KUKA KRL program: Milling_8_3.src

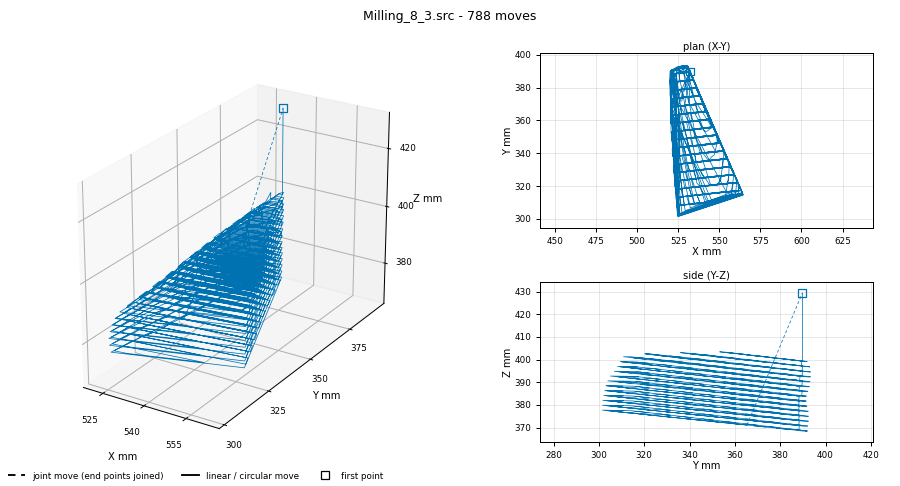
[picture p0: tool path of Milling_8_3.src, 788 of 790 moves have a stored position in this frame; points joined in program order, loops and branches not executed]
&ACCESS RVP
&REL 1
&PARAM TEMPLATE = C:\KRC\Roboter\Template\vorgabe
&PARAM EDITMASK = *
DEF Milling_8_3 ( )


;FOLD INI
;FOLD BASISTECH INI
GLOBAL INTERRUPT DECL 3 WHEN $STOPMESS==TRUE DO IR_STOPM ( )
INTERRUPT ON 3
BAS (#INITMOV,0 )
;ENDFOLD (BASISTECH INI)
;ENDFOLD (INI)

;FOLD STARTPOSITION - BASE IS 0, TOOL IS 5, SPEED IS 15%, POSITION IS A1 5,A2 -90,A3 100,A4 5,A5 -10,A6 -5,E1 0,E2 0,E3 0,E4 0
$BWDSTART = FALSE
PDAT_ACT = {VEL 15,ACC 100,APO_DIST 50}
FDAT_ACT = {TOOL_NO 5,BASE_NO 0,IPO_FRAME #BASE}
BAS (#PTP_PARAMS,15)
PTP  {A1 5,A2 -90,A3 100,A4 5,A5 -10,A6 -5,E1 0,E2 0,E3 0,E4 0}
;ENDFOLD

;FOLD LIN SPEED IS 0.1 m/sec, INTERPOLATION SETTINGS IN FOLD
$VEL.CP=0.1
$ADVANCE=3
;ENDFOLD

BAS(#VEL_PTP,2)
PTP {X 532.274, Y 389.769, Z 429.374, A -75.058, B 83.904, C 170.36, E1 0, E2 0, E3 0, E4 0, S 'B010'}
$VEL.CP=0.012
LIN {X 532.274, Y 389.769, Z 399.374, A -75.058, B 83.904, C 170.36, E1 0, E2 0, E3 0, E4 0}
LIN {X 530.976, Y 389.628, Z 399.353, A -75.058, B 83.904, C 170.36, E1 0, E2 0, E3 0, E4 0}
LIN {X 531.862, Y 384.703, Z 399.885, A -75.058, B 83.904, C 170.36, E1 0, E2 0, E3 0, E4 0}
LIN {X 534.21, Y 384.958, Z 399.924, A -75.058, B 83.904, C 170.36, E1 0, E2 0, E3 0, E4 0}
LIN {X 536.146, Y 380.148, Z 400.473, A -75.058, B 83.904, C 170.36, E1 0, E2 0, E3 0, E4 0}
LIN {X 532.732, Y 379.777, Z 400.418, A -75.058, B 83.904, C 170.36, E1 0, E2 0, E3 0, E4 0}
LIN {X 533.878, Y 374.881, Z 400.954, A -75.058, B 83.904, C 170.36, E1 0, E2 0, E3 0, E4 0}
LIN {X 538.082, Y 375.337, Z 401.023, A -75.058, B 83.904, C 170.36, E1 0, E2 0, E3 0, E4 0}
LIN {X 540.018, Y 370.527, Z 401.573, A -75.058, B 83.904, C 170.36, E1 0, E2 0, E3 0, E4 0}
LIN {X 535.26, Y 370.011, Z 401.495, A -75.058, B 83.904, C 170.36, E1 0, E2 0, E3 0, E4 0}
LIN {X 536.788, Y 365.156, Z 402.038, A -75.058, B 83.904, C 170.36, E1 0, E2 0, E3 0, E4 0}
LIN {X 541.954, Y 365.716, Z 402.123, A -75.058, B 83.904, C 170.36, E1 0, E2 0, E3 0, E4 0}
LIN {X 544.073, Y 360.926, Z 402.675, A -75.058, B 83.904, C 170.36, E1 0, E2 0, E3 0, E4 0}
LIN {X 538.348, Y 360.305, Z 402.582, A -75.058, B 83.904, C 170.36, E1 0, E2 0, E3 0, E4 0}
LIN {X 539.977, Y 355.461, Z 403.126, A -75.058, B 83.904, C 170.36, E1 0, E2 0, E3 0, E4 0}
LIN {X 545.351, Y 356.044, Z 403.214, A -75.058, B 83.904, C 170.36, E1 0, E2 0, E3 0, E4 0}
LIN {X 535.132, Y 372.263, Z 401.259, A -75.058, B 83.904, C 170.36, E1 0, E2 0, E3 0, E4 0}
LIN {X 537.332, Y 363.753, Z 402.198, A -75.058, B 83.904, C 170.36, E1 0, E2 0, E3 0, E4 0}
LIN {X 537.362, Y 363.721, Z 402.202, A -75.058, B 83.904, C 170.36, E1 0, E2 0, E3 0, E4 0}
LIN {X 538.426, Y 361.065, Z 402.505, A -75.058, B 83.904, C 170.36, E1 0, E2 0, E3 0, E4 0}
LIN {X 538.125, Y 359.587, Z 402.65, A -75.058, B 83.904, C 170.36, E1 0, E2 0, E3 0, E4 0}
LIN {X 538.164, Y 358.226, Z 402.791, A -75.058, B 83.904, C 170.36, E1 0, E2 0, E3 0, E4 0}
LIN {X 538.673, Y 356.747, Z 402.958, A -75.058, B 83.904, C 170.36, E1 0, E2 0, E3 0, E4 0}
LIN {X 540.02, Y 355.418, Z 403.132, A -75.058, B 83.904, C 170.36, E1 0, E2 0, E3 0, E4 0}
LIN {X 540.271, Y 354.332, Z 403.251, A -75.058, B 83.904, C 170.36, E1 0, E2 0, E3 0, E4 0}
LIN {X 540.872, Y 353.577, Z 403.345, A -75.058, B 83.904, C 170.36, E1 0, E2 0, E3 0, E4 0}
LIN {X 541.194, Y 353.443, Z 403.368, A -75.058, B 83.904, C 170.36, E1 0, E2 0, E3 0, E4 0}
LIN {X 542.255, Y 353.309, Z 403.411, A -75.058, B 83.904, C 170.36, E1 0, E2 0, E3 0, E4 0}
LIN {X 542.693, Y 353.497, Z 403.404, A -75.058, B 83.904, C 170.36, E1 0, E2 0, E3 0, E4 0}
LIN {X 545.139, Y 355.6, Z 403.254, A -75.058, B 83.904, C 170.36, E1 0, E2 0, E3 0, E4 0}
LIN {X 545.858, Y 356.987, Z 403.131, A -75.058, B 83.904, C 170.36, E1 0, E2 0, E3 0, E4 0}
LIN {X 531.417, Y 391.899, Z 399.131, A -75.058, B 83.904, C 170.36, E1 0, E2 0, E3 0, E4 0}
LIN {X 531.262, Y 391.678, Z 399.149, A -75.058, B 83.904, C 170.36, E1 0, E2 0, E3 0, E4 0}
LIN {X 530.896, Y 390.596, Z 399.251, A -75.058, B 83.904, C 170.36, E1 0, E2 0, E3 0, E4 0}
LIN {X 531.291, Y 387.123, Z 399.62, A -75.058, B 83.904, C 170.36, E1 0, E2 0, E3 0, E4 0}
LIN {X 535.132, Y 372.263, Z 401.259, A -75.058, B 83.904, C 170.36, E1 0, E2 0, E3 0, E4 0}
LIN {X 528.021, Y 389.496, Z 399.285, A -75.058, B 83.904, C 170.36, E1 0, E2 0, E3 0, E4 0}
LIN {X 528.08, Y 389.273, Z 397.124, A -75.058, B 83.904, C 170.36, E1 0, E2 0, E3 0, E4 0}
LIN {X 532.261, Y 389.727, Z 397.192, A -75.058, B 83.904, C 170.36, E1 0, E2 0, E3 0, E4 0}
LIN {X 534.197, Y 384.916, Z 397.741, A -75.058, B 83.904, C 170.36, E1 0, E2 0, E3 0, E4 0}
LIN {X 528.642, Y 384.314, Z 397.651, A -75.058, B 83.904, C 170.36, E1 0, E2 0, E3 0, E4 0}
LIN {X 529.632, Y 379.401, Z 398.185, A -75.058, B 83.904, C 170.36, E1 0, E2 0, E3 0, E4 0}
LIN {X 536.133, Y 380.106, Z 398.291, A -75.058, B 83.904, C 170.36, E1 0, E2 0, E3 0, E4 0}
LIN {X 538.069, Y 375.295, Z 398.841, A -75.058, B 83.904, C 170.36, E1 0, E2 0, E3 0, E4 0}
LIN {X 530.533, Y 374.478, Z 398.718, A -75.058, B 83.904, C 170.36, E1 0, E2 0, E3 0, E4 0}
LIN {X 531.748, Y 369.589, Z 399.256, A -75.058, B 83.904, C 170.36, E1 0, E2 0, E3 0, E4 0}
LIN {X 540.005, Y 370.485, Z 399.39, A -75.058, B 83.904, C 170.36, E1 0, E2 0, E3 0, E4 0}
LIN {X 541.941, Y 365.674, Z 399.94, A -75.058, B 83.904, C 170.36, E1 0, E2 0, E3 0, E4 0}
LIN {X 532.254, Y 364.624, Z 399.782, A -75.058, B 83.904, C 170.36, E1 0, E2 0, E3 0, E4 0}
LIN {X 533.519, Y 359.741, Z 400.321, A -75.058, B 83.904, C 170.36, E1 0, E2 0, E3 0, E4 0}
LIN {X 544.051, Y 360.883, Z 400.493, A -75.058, B 83.904, C 170.36, E1 0, E2 0, E3 0, E4 0}
LIN {X 546.219, Y 356.098, Z 401.046, A -75.058, B 83.904, C 170.36, E1 0, E2 0, E3 0, E4 0}
LIN {X 534.728, Y 354.851, Z 400.858, A -75.058, B 83.904, C 170.36, E1 0, E2 0, E3 0, E4 0}
LIN {X 535.946, Y 349.963, Z 401.396, A -75.058, B 83.904, C 170.36, E1 0, E2 0, E3 0, E4 0}
LIN {X 548.387, Y 351.312, Z 401.6, A -75.058, B 83.904, C 170.36, E1 0, E2 0, E3 0, E4 0}
LIN {X 548.738, Y 346.33, Z 402.123, A -75.058, B 83.904, C 170.36, E1 0, E2 0, E3 0, E4 0}
LIN {X 537.964, Y 345.161, Z 401.947, A -75.058, B 83.904, C 170.36, E1 0, E2 0, E3 0, E4 0}
LIN {X 539.662, Y 340.325, Z 402.493, A -75.058, B 83.904, C 170.36, E1 0, E2 0, E3 0, E4 0}
LIN {X 547.662, Y 341.193, Z 402.624, A -75.058, B 83.904, C 170.36, E1 0, E2 0, E3 0, E4 0}
LIN {X 531.803, Y 370.273, Z 399.187, A -75.058, B 83.904, C 170.36, E1 0, E2 0, E3 0, E4 0}
LIN {X 534.557, Y 355.635, Z 400.773, A -75.058, B 83.904, C 170.36, E1 0, E2 0, E3 0, E4 0}
LIN {X 535.012, Y 351.656, Z 401.196, A -75.058, B 83.904, C 170.36, E1 0, E2 0, E3 0, E4 0}
LIN {X 539.065, Y 341.32, Z 402.374, A -75.058, B 83.904, C 170.36, E1 0, E2 0, E3 0, E4 0}
LIN {X 543.057, Y 336.009, Z 403.032, A -75.058, B 83.904, C 170.36, E1 0, E2 0, E3 0, E4 0}
LIN {X 544.101, Y 336.271, Z 403.034, A -75.058, B 83.904, C 170.36, E1 0, E2 0, E3 0, E4 0}
LIN {X 545.466, Y 337.952, Z 402.898, A -75.058, B 83.904, C 170.36, E1 0, E2 0, E3 0, E4 0}
LIN {X 546.771, Y 338.821, Z 402.844, A -75.058, B 83.904, C 170.36, E1 0, E2 0, E3 0, E4 0}
LIN {X 546.979, Y 339.189, Z 402.812, A -75.058, B 83.904, C 170.36, E1 0, E2 0, E3 0, E4 0}
LIN {X 549.393, Y 349.092, Z 401.856, A -75.058, B 83.904, C 170.36, E1 0, E2 0, E3 0, E4 0}
LIN {X 530.975, Y 392.923, Z 396.827, A -75.058, B 83.904, C 170.36, E1 0, E2 0, E3 0, E4 0}
LIN {X 530.15, Y 392.664, Z 396.831, A -75.058, B 83.904, C 170.36, E1 0, E2 0, E3 0, E4 0}
LIN {X 529.187, Y 392.933, Z 396.776, A -75.058, B 83.904, C 170.36, E1 0, E2 0, E3 0, E4 0}
LIN {X 528.673, Y 392.74, Z 396.782, A -75.058, B 83.904, C 170.36, E1 0, E2 0, E3 0, E4 0}
LIN {X 528.244, Y 391.836, Z 396.864, A -75.058, B 83.904, C 170.36, E1 0, E2 0, E3 0, E4 0}
LIN {X 528.038, Y 390.278, Z 397.019, A -75.058, B 83.904, C 170.36, E1 0, E2 0, E3 0, E4 0}
LIN {X 531.803, Y 370.273, Z 399.187, A -75.058, B 83.904, C 170.36, E1 0, E2 0, E3 0, E4 0}
LIN {X 532.188, Y 389.908, Z 397.171, A -75.058, B 83.904, C 170.36, E1 0, E2 0, E3 0, E4 0}
LIN {X 532.247, Y 389.685, Z 395.01, A -75.058, B 83.904, C 170.36, E1 0, E2 0, E3 0, E4 0}
LIN {X 525.532, Y 388.957, Z 394.9, A -75.058, B 83.904, C 170.36, E1 0, E2 0, E3 0, E4 0}
LIN {X 525.92, Y 383.978, Z 395.424, A -75.058, B 83.904, C 170.36, E1 0, E2 0, E3 0, E4 0}
LIN {X 534.183, Y 384.875, Z 395.559, A -75.058, B 83.904, C 170.36, E1 0, E2 0, E3 0, E4 0}
LIN {X 536.119, Y 380.064, Z 396.109, A -75.058, B 83.904, C 170.36, E1 0, E2 0, E3 0, E4 0}
LIN {X 526.867, Y 379.061, Z 395.958, A -75.058, B 83.904, C 170.36, E1 0, E2 0, E3 0, E4 0}
LIN {X 527.599, Y 374.12, Z 396.488, A -75.058, B 83.904, C 170.36, E1 0, E2 0, E3 0, E4 0}
LIN {X 538.055, Y 375.254, Z 396.659, A -75.058, B 83.904, C 170.36, E1 0, E2 0, E3 0, E4 0}
LIN {X 539.991, Y 370.443, Z 397.208, A -75.058, B 83.904, C 170.36, E1 0, E2 0, E3 0, E4 0}
LIN {X 528.317, Y 369.177, Z 397.017, A -75.058, B 83.904, C 170.36, E1 0, E2 0, E3 0, E4 0}
LIN {X 529.23, Y 364.256, Z 397.55, A -75.058, B 83.904, C 170.36, E1 0, E2 0, E3 0, E4 0}
LIN {X 541.927, Y 365.633, Z 397.758, A -75.058, B 83.904, C 170.36, E1 0, E2 0, E3 0, E4 0}
LIN {X 544.029, Y 360.84, Z 398.31, A -75.058, B 83.904, C 170.36, E1 0, E2 0, E3 0, E4 0}
LIN {X 529.983, Y 359.317, Z 398.081, A -75.058, B 83.904, C 170.36, E1 0, E2 0, E3 0, E4 0}
LIN {X 531.088, Y 354.416, Z 398.617, A -75.058, B 83.904, C 170.36, E1 0, E2 0, E3 0, E4 0}
LIN {X 546.197, Y 356.055, Z 398.864, A -75.058, B 83.904, C 170.36, E1 0, E2 0, E3 0, E4 0}
LIN {X 548.365, Y 351.27, Z 399.417, A -75.058, B 83.904, C 170.36, E1 0, E2 0, E3 0, E4 0}
LIN {X 532.342, Y 349.532, Z 399.155, A -75.058, B 83.904, C 170.36, E1 0, E2 0, E3 0, E4 0}
LIN {X 533.594, Y 344.647, Z 399.694, A -75.058, B 83.904, C 170.36, E1 0, E2 0, E3 0, E4 0}
LIN {X 550.532, Y 346.484, Z 399.971, A -75.058, B 83.904, C 170.36, E1 0, E2 0, E3 0, E4 0}
LIN {X 552.698, Y 341.699, Z 400.524, A -75.058, B 83.904, C 170.36, E1 0, E2 0, E3 0, E4 0}
LIN {X 534.899, Y 339.768, Z 400.233, A -75.058, B 83.904, C 170.36, E1 0, E2 0, E3 0, E4 0}
LIN {X 535.865, Y 334.853, Z 400.767, A -75.058, B 83.904, C 170.36, E1 0, E2 0, E3 0, E4 0}
LIN {X 552.362, Y 336.642, Z 401.037, A -75.058, B 83.904, C 170.36, E1 0, E2 0, E3 0, E4 0}
LIN {X 552.046, Y 331.587, Z 401.55, A -75.058, B 83.904, C 170.36, E1 0, E2 0, E3 0, E4 0}
LIN {X 538.149, Y 330.08, Z 401.322, A -75.058, B 83.904, C 170.36, E1 0, E2 0, E3 0, E4 0}
LIN {X 540.909, Y 325.359, Z 401.885, A -75.058, B 83.904, C 170.36, E1 0, E2 0, E3 0, E4 0}
LIN {X 551.401, Y 326.497, Z 402.057, A -75.058, B 83.904, C 170.36, E1 0, E2 0, E3 0, E4 0}
LIN {X 549.185, Y 321.236, Z 402.539, A -75.058, B 83.904, C 170.36, E1 0, E2 0, E3 0, E4 0}
LIN {X 544.732, Y 320.753, Z 402.466, A -75.058, B 83.904, C 170.36, E1 0, E2 0, E3 0, E4 0}
LIN {X 529.043, Y 369.622, Z 396.991, A -75.058, B 83.904, C 170.36, E1 0, E2 0, E3 0, E4 0}
LIN {X 535.031, Y 339.499, Z 400.264, A -75.058, B 83.904, C 170.36, E1 0, E2 0, E3 0, E4 0}
LIN {X 535.862, Y 334.867, Z 400.765, A -75.058, B 83.904, C 170.36, E1 0, E2 0, E3 0, E4 0}
LIN {X 539.532, Y 326.865, Z 401.692, A -75.058, B 83.904, C 170.36, E1 0, E2 0, E3 0, E4 0}
LIN {X 541.886, Y 324.365, Z 402.015, A -75.058, B 83.904, C 170.36, E1 0, E2 0, E3 0, E4 0}
LIN {X 541.983, Y 323.772, Z 402.079, A -75.058, B 83.904, C 170.36, E1 0, E2 0, E3 0, E4 0}
LIN {X 542.174, Y 323.744, Z 402.087, A -75.058, B 83.904, C 170.36, E1 0, E2 0, E3 0, E4 0}
LIN {X 543.943, Y 321.055, Z 402.413, A -75.058, B 83.904, C 170.36, E1 0, E2 0, E3 0, E4 0}
LIN {X 546.874, Y 320.282, Z 402.574, A -75.058, B 83.904, C 170.36, E1 0, E2 0, E3 0, E4 0}
LIN {X 549.787, Y 321.563, Z 402.522, A -75.058, B 83.904, C 170.36, E1 0, E2 0, E3 0, E4 0}
LIN {X 549.819, Y 321.567, Z 402.522, A -75.058, B 83.904, C 170.36, E1 0, E2 0, E3 0, E4 0}
LIN {X 550.895, Y 323.874, Z 402.314, A -75.058, B 83.904, C 170.36, E1 0, E2 0, E3 0, E4 0}
LIN {X 552.942, Y 341.161, Z 400.586, A -75.058, B 83.904, C 170.36, E1 0, E2 0, E3 0, E4 0}
LIN {X 530.976, Y 392.844, Z 394.649, A -75.058, B 83.904, C 170.36, E1 0, E2 0, E3 0, E4 0}
LIN {X 530.18, Y 392.7, Z 394.641, A -75.058, B 83.904, C 170.36, E1 0, E2 0, E3 0, E4 0}
LIN {X 529.535, Y 393.045, Z 394.588, A -75.058, B 83.904, C 170.36, E1 0, E2 0, E3 0, E4 0}
LIN {X 527.957, Y 393.376, Z 394.51, A -75.058, B 83.904, C 170.36, E1 0, E2 0, E3 0, E4 0}
LIN {X 526.259, Y 392.781, Z 394.525, A -75.058, B 83.904, C 170.36, E1 0, E2 0, E3 0, E4 0}
LIN {X 526.107, Y 392.584, Z 394.541, A -75.058, B 83.904, C 170.36, E1 0, E2 0, E3 0, E4 0}
LIN {X 525.559, Y 387.147, Z 395.087, A -75.058, B 83.904, C 170.36, E1 0, E2 0, E3 0, E4 0}
LIN {X 529.043, Y 369.622, Z 396.991, A -75.058, B 83.904, C 170.36, E1 0, E2 0, E3 0, E4 0}
LIN {X 532.174, Y 389.866, Z 394.989, A -75.058, B 83.904, C 170.36, E1 0, E2 0, E3 0, E4 0}
LIN {X 532.234, Y 389.643, Z 392.827, A -75.058, B 83.904, C 170.36, E1 0, E2 0, E3 0, E4 0}
LIN {X 523.817, Y 388.731, Z 392.689, A -75.058, B 83.904, C 170.36, E1 0, E2 0, E3 0, E4 0}
LIN {X 523.955, Y 383.725, Z 393.21, A -75.058, B 83.904, C 170.36, E1 0, E2 0, E3 0, E4 0}
LIN {X 534.17, Y 384.833, Z 393.377, A -75.058, B 83.904, C 170.36, E1 0, E2 0, E3 0, E4 0}
LIN {X 536.106, Y 380.022, Z 393.926, A -75.058, B 83.904, C 170.36, E1 0, E2 0, E3 0, E4 0}
LIN {X 524.629, Y 378.777, Z 393.739, A -75.058, B 83.904, C 170.36, E1 0, E2 0, E3 0, E4 0}
LIN {X 525.426, Y 373.844, Z 394.27, A -75.058, B 83.904, C 170.36, E1 0, E2 0, E3 0, E4 0}
LIN {X 538.042, Y 375.212, Z 394.476, A -75.058, B 83.904, C 170.36, E1 0, E2 0, E3 0, E4 0}
LIN {X 539.978, Y 370.401, Z 395.026, A -75.058, B 83.904, C 170.36, E1 0, E2 0, E3 0, E4 0}
LIN {X 526.195, Y 368.907, Z 394.801, A -75.058, B 83.904, C 170.36, E1 0, E2 0, E3 0, E4 0}
LIN {X 527.04, Y 363.978, Z 395.332, A -75.058, B 83.904, C 170.36, E1 0, E2 0, E3 0, E4 0}
LIN {X 541.914, Y 365.591, Z 395.576, A -75.058, B 83.904, C 170.36, E1 0, E2 0, E3 0, E4 0}
LIN {X 544.007, Y 360.798, Z 396.128, A -75.058, B 83.904, C 170.36, E1 0, E2 0, E3 0, E4 0}
LIN {X 527.523, Y 359.01, Z 395.858, A -75.058, B 83.904, C 170.36, E1 0, E2 0, E3 0, E4 0}
LIN {X 528.524, Y 354.098, Z 396.393, A -75.058, B 83.904, C 170.36, E1 0, E2 0, E3 0, E4 0}
LIN {X 546.175, Y 356.012, Z 396.681, A -75.058, B 83.904, C 170.36, E1 0, E2 0, E3 0, E4 0}
LIN {X 548.343, Y 351.227, Z 397.235, A -75.058, B 83.904, C 170.36, E1 0, E2 0, E3 0, E4 0}
LIN {X 529.958, Y 349.233, Z 396.934, A -75.058, B 83.904, C 170.36, E1 0, E2 0, E3 0, E4 0}
LIN {X 530.947, Y 344.32, Z 397.468, A -75.058, B 83.904, C 170.36, E1 0, E2 0, E3 0, E4 0}
LIN {X 550.511, Y 346.442, Z 397.788, A -75.058, B 83.904, C 170.36, E1 0, E2 0, E3 0, E4 0}
LIN {X 552.679, Y 341.656, Z 398.342, A -75.058, B 83.904, C 170.36, E1 0, E2 0, E3 0, E4 0}
LIN {X 532.163, Y 339.431, Z 398.006, A -75.058, B 83.904, C 170.36, E1 0, E2 0, E3 0, E4 0}
LIN {X 533.107, Y 334.513, Z 398.54, A -75.058, B 83.904, C 170.36, E1 0, E2 0, E3 0, E4 0}
LIN {X 554.847, Y 336.871, Z 398.895, A -75.058, B 83.904, C 170.36, E1 0, E2 0, E3 0, E4 0}
LIN {X 556.033, Y 331.979, Z 399.433, A -75.058, B 83.904, C 170.36, E1 0, E2 0, E3 0, E4 0}
LIN {X 534.262, Y 329.618, Z 399.077, A -75.058, B 83.904, C 170.36, E1 0, E2 0, E3 0, E4 0}
LIN {X 535.701, Y 324.754, Z 399.618, A -75.058, B 83.904, C 170.36, E1 0, E2 0, E3 0, E4 0}
LIN {X 555.87, Y 326.941, Z 399.948, A -75.058, B 83.904, C 170.36, E1 0, E2 0, E3 0, E4 0}
LIN {X 554.99, Y 321.825, Z 400.451, A -75.058, B 83.904, C 170.36, E1 0, E2 0, E3 0, E4 0}
LIN {X 537.868, Y 319.968, Z 400.172, A -75.058, B 83.904, C 170.36, E1 0, E2 0, E3 0, E4 0}
LIN {X 540.443, Y 315.227, Z 400.732, A -75.058, B 83.904, C 170.36, E1 0, E2 0, E3 0, E4 0}
LIN {X 554.164, Y 316.715, Z 400.956, A -75.058, B 83.904, C 170.36, E1 0, E2 0, E3 0, E4 0}
LIN {X 526.44, Y 368.431, Z 394.856, A -75.058, B 83.904, C 170.36, E1 0, E2 0, E3 0, E4 0}
LIN {X 527.197, Y 362.973, Z 395.44, A -75.058, B 83.904, C 170.36, E1 0, E2 0, E3 0, E4 0}
LIN {X 536.476, Y 321.636, Z 399.961, A -75.058, B 83.904, C 170.36, E1 0, E2 0, E3 0, E4 0}
LIN {X 537.55, Y 320.622, Z 400.095, A -75.058, B 83.904, C 170.36, E1 0, E2 0, E3 0, E4 0}
LIN {X 540.97, Y 314.37, Z 400.835, A -75.058, B 83.904, C 170.36, E1 0, E2 0, E3 0, E4 0}
LIN {X 541.552, Y 312.236, Z 401.071, A -75.058, B 83.904, C 170.36, E1 0, E2 0, E3 0, E4 0}
LIN {X 542.631, Y 310.895, Z 401.239, A -75.058, B 83.904, C 170.36, E1 0, E2 0, E3 0, E4 0}
LIN {X 553.838, Y 314.095, Z 401.217, A -75.058, B 83.904, C 170.36, E1 0, E2 0, E3 0, E4 0}
LIN {X 554.994, Y 321.94, Z 400.44, A -75.058, B 83.904, C 170.36, E1 0, E2 0, E3 0, E4 0}
LIN {X 555.677, Y 323.872, Z 400.259, A -75.058, B 83.904, C 170.36, E1 0, E2 0, E3 0, E4 0}
LIN {X 555.938, Y 332.724, Z 399.353, A -75.058, B 83.904, C 170.36, E1 0, E2 0, E3 0, E4 0}
LIN {X 556.034, Y 334.252, Z 399.198, A -75.058, B 83.904, C 170.36, E1 0, E2 0, E3 0, E4 0}
LIN {X 530.801, Y 393.204, Z 392.42, A -75.058, B 83.904, C 170.36, E1 0, E2 0, E3 0, E4 0}
LIN {X 529.984, Y 393.067, Z 392.412, A -75.058, B 83.904, C 170.36, E1 0, E2 0, E3 0, E4 0}
LIN {X 527.427, Y 393.254, Z 392.322, A -75.058, B 83.904, C 170.36, E1 0, E2 0, E3 0, E4 0}
LIN {X 524.679, Y 392.5, Z 392.324, A -75.058, B 83.904, C 170.36, E1 0, E2 0, E3 0, E4 0}
LIN {X 524.141, Y 391.998, Z 392.361, A -75.058, B 83.904, C 170.36, E1 0, E2 0, E3 0, E4 0}
LIN {X 523.784, Y 391.286, Z 392.425, A -75.058, B 83.904, C 170.36, E1 0, E2 0, E3 0, E4 0}
LIN {X 523.836, Y 387.741, Z 392.792, A -75.058, B 83.904, C 170.36, E1 0, E2 0, E3 0, E4 0}
LIN {X 523.78, Y 387.627, Z 392.802, A -75.058, B 83.904, C 170.36, E1 0, E2 0, E3 0, E4 0}
LIN {X 526.44, Y 368.431, Z 394.856, A -75.058, B 83.904, C 170.36, E1 0, E2 0, E3 0, E4 0}
LIN {X 522.26, Y 388.751, Z 392.645, A -75.058, B 83.904, C 170.36, E1 0, E2 0, E3 0, E4 0}
LIN {X 522.32, Y 388.528, Z 390.483, A -75.058, B 83.904, C 170.36, E1 0, E2 0, E3 0, E4 0}
LIN {X 532.221, Y 389.602, Z 390.645, A -75.058, B 83.904, C 170.36, E1 0, E2 0, E3 0, E4 0}
LIN {X 534.157, Y 384.791, Z 391.195, A -75.058, B 83.904, C 170.36, E1 0, E2 0, E3 0, E4 0}
LIN {X 522.238, Y 383.499, Z 391, A -75.058, B 83.904, C 170.36, E1 0, E2 0, E3 0, E4 0}
LIN {X 522.794, Y 378.538, Z 391.527, A -75.058, B 83.904, C 170.36, E1 0, E2 0, E3 0, E4 0}
LIN {X 536.093, Y 379.981, Z 391.744, A -75.058, B 83.904, C 170.36, E1 0, E2 0, E3 0, E4 0}
LIN {X 538.028, Y 375.17, Z 392.294, A -75.058, B 83.904, C 170.36, E1 0, E2 0, E3 0, E4 0}
LIN {X 523.48, Y 373.592, Z 392.056, A -75.058, B 83.904, C 170.36, E1 0, E2 0, E3 0, E4 0}
LIN {X 524.317, Y 368.663, Z 392.588, A -75.058, B 83.904, C 170.36, E1 0, E2 0, E3 0, E4 0}
LIN {X 539.964, Y 370.36, Z 392.843, A -75.058, B 83.904, C 170.36, E1 0, E2 0, E3 0, E4 0}
LIN {X 541.9, Y 365.549, Z 393.393, A -75.058, B 83.904, C 170.36, E1 0, E2 0, E3 0, E4 0}
LIN {X 525.071, Y 363.724, Z 393.118, A -75.058, B 83.904, C 170.36, E1 0, E2 0, E3 0, E4 0}
LIN {X 525.771, Y 358.779, Z 393.648, A -75.058, B 83.904, C 170.36, E1 0, E2 0, E3 0, E4 0}
LIN {X 543.985, Y 360.755, Z 393.945, A -75.058, B 83.904, C 170.36, E1 0, E2 0, E3 0, E4 0}
LIN {X 546.153, Y 355.97, Z 394.499, A -75.058, B 83.904, C 170.36, E1 0, E2 0, E3 0, E4 0}
LIN {X 526.266, Y 353.813, Z 394.174, A -75.058, B 83.904, C 170.36, E1 0, E2 0, E3 0, E4 0}
LIN {X 527.416, Y 348.917, Z 394.711, A -75.058, B 83.904, C 170.36, E1 0, E2 0, E3 0, E4 0}
LIN {X 548.321, Y 351.184, Z 395.052, A -75.058, B 83.904, C 170.36, E1 0, E2 0, E3 0, E4 0}
LIN {X 550.489, Y 346.399, Z 395.606, A -75.058, B 83.904, C 170.36, E1 0, E2 0, E3 0, E4 0}
LIN {X 528.352, Y 343.998, Z 395.244, A -75.058, B 83.904, C 170.36, E1 0, E2 0, E3 0, E4 0}
LIN {X 529.601, Y 339.113, Z 395.782, A -75.058, B 83.904, C 170.36, E1 0, E2 0, E3 0, E4 0}
LIN {X 552.657, Y 341.614, Z 396.159, A -75.058, B 83.904, C 170.36, E1 0, E2 0, E3 0, E4 0}
LIN {X 554.825, Y 336.828, Z 396.713, A -75.058, B 83.904, C 170.36, E1 0, E2 0, E3 0, E4 0}
LIN {X 530.607, Y 334.202, Z 396.317, A -75.058, B 83.904, C 170.36, E1 0, E2 0, E3 0, E4 0}
LIN {X 531.871, Y 329.318, Z 396.855, A -75.058, B 83.904, C 170.36, E1 0, E2 0, E3 0, E4 0}
LIN {X 556.993, Y 332.043, Z 397.266, A -75.058, B 83.904, C 170.36, E1 0, E2 0, E3 0, E4 0}
LIN {X 558.925, Y 327.232, Z 397.816, A -75.058, B 83.904, C 170.36, E1 0, E2 0, E3 0, E4 0}
LIN {X 532.872, Y 324.407, Z 397.39, A -75.058, B 83.904, C 170.36, E1 0, E2 0, E3 0, E4 0}
LIN {X 534.194, Y 319.529, Z 397.93, A -75.058, B 83.904, C 170.36, E1 0, E2 0, E3 0, E4 0}
LIN {X 558.615, Y 322.178, Z 398.329, A -75.058, B 83.904, C 170.36, E1 0, E2 0, E3 0, E4 0}
LIN {X 557.516, Y 317.039, Z 398.829, A -75.058, B 83.904, C 170.36, E1 0, E2 0, E3 0, E4 0}
LIN {X 536.361, Y 314.744, Z 398.483, A -75.058, B 83.904, C 170.36, E1 0, E2 0, E3 0, E4 0}
LIN {X 538.149, Y 309.918, Z 399.03, A -75.058, B 83.904, C 170.36, E1 0, E2 0, E3 0, E4 0}
LIN {X 541.212, Y 310.25, Z 399.08, A -75.058, B 83.904, C 170.36, E1 0, E2 0, E3 0, E4 0}
LIN {X 524.865, Y 368.056, Z 392.665, A -75.058, B 83.904, C 170.36, E1 0, E2 0, E3 0, E4 0}
LIN {X 528.337, Y 345.247, Z 395.115, A -75.058, B 83.904, C 170.36, E1 0, E2 0, E3 0, E4 0}
LIN {X 528.352, Y 343.922, Z 395.252, A -75.058, B 83.904, C 170.36, E1 0, E2 0, E3 0, E4 0}
LIN {X 529.108, Y 341.583, Z 395.514, A -75.058, B 83.904, C 170.36, E1 0, E2 0, E3 0, E4 0}
LIN {X 530.622, Y 333.185, Z 396.422, A -75.058, B 83.904, C 170.36, E1 0, E2 0, E3 0, E4 0}
LIN {X 536.653, Y 314.101, Z 398.557, A -75.058, B 83.904, C 170.36, E1 0, E2 0, E3 0, E4 0}
LIN {X 536.673, Y 313.884, Z 398.58, A -75.058, B 83.904, C 170.36, E1 0, E2 0, E3 0, E4 0}
LIN {X 538.421, Y 309.453, Z 399.086, A -75.058, B 83.904, C 170.36, E1 0, E2 0, E3 0, E4 0}
LIN {X 557.231, Y 314.824, Z 399.049, A -75.058, B 83.904, C 170.36, E1 0, E2 0, E3 0, E4 0}
LIN {X 558.944, Y 327.737, Z 397.764, A -75.058, B 83.904, C 170.36, E1 0, E2 0, E3 0, E4 0}
LIN {X 530.778, Y 393.188, Z 390.235, A -75.058, B 83.904, C 170.36, E1 0, E2 0, E3 0, E4 0}
LIN {X 529.944, Y 393.172, Z 390.214, A -75.058, B 83.904, C 170.36, E1 0, E2 0, E3 0, E4 0}
LIN {X 523.929, Y 392.372, Z 390.131, A -75.058, B 83.904, C 170.36, E1 0, E2 0, E3 0, E4 0}
LIN {X 523.089, Y 391.847, Z 390.162, A -75.058, B 83.904, C 170.36, E1 0, E2 0, E3 0, E4 0}
LIN {X 522.749, Y 391.345, Z 390.204, A -75.058, B 83.904, C 170.36, E1 0, E2 0, E3 0, E4 0}
LIN {X 521.947, Y 387.325, Z 390.597, A -75.058, B 83.904, C 170.36, E1 0, E2 0, E3 0, E4 0}
LIN {X 521.962, Y 386.746, Z 390.657, A -75.058, B 83.904, C 170.36, E1 0, E2 0, E3 0, E4 0}
LIN {X 522.034, Y 386.649, Z 390.669, A -75.058, B 83.904, C 170.36, E1 0, E2 0, E3 0, E4 0}
LIN {X 524.865, Y 368.056, Z 392.665, A -75.058, B 83.904, C 170.36, E1 0, E2 0, E3 0, E4 0}
LIN {X 532.148, Y 389.783, Z 390.624, A -75.058, B 83.904, C 170.36, E1 0, E2 0, E3 0, E4 0}
LIN {X 532.207, Y 389.56, Z 388.462, A -75.058, B 83.904, C 170.36, E1 0, E2 0, E3 0, E4 0}
LIN {X 520.886, Y 388.332, Z 388.277, A -75.058, B 83.904, C 170.36, E1 0, E2 0, E3 0, E4 0}
LIN {X 520.772, Y 383.299, Z 388.794, A -75.058, B 83.904, C 170.36, E1 0, E2 0, E3 0, E4 0}
LIN {X 534.143, Y 384.749, Z 389.012, A -75.058, B 83.904, C 170.36, E1 0, E2 0, E3 0, E4 0}
LIN {X 536.079, Y 379.939, Z 389.562, A -75.058, B 83.904, C 170.36, E1 0, E2 0, E3 0, E4 0}
LIN {X 521.403, Y 378.347, Z 389.322, A -75.058, B 83.904, C 170.36, E1 0, E2 0, E3 0, E4 0}
LIN {X 522.109, Y 373.403, Z 389.851, A -75.058, B 83.904, C 170.36, E1 0, E2 0, E3 0, E4 0}
LIN {X 538.015, Y 375.128, Z 390.111, A -75.058, B 83.904, C 170.36, E1 0, E2 0, E3 0, E4 0}
LIN {X 539.951, Y 370.318, Z 390.661, A -75.058, B 83.904, C 170.36, E1 0, E2 0, E3 0, E4 0}
LIN {X 522.685, Y 368.445, Z 390.379, A -75.058, B 83.904, C 170.36, E1 0, E2 0, E3 0, E4 0}
LIN {X 523.359, Y 363.498, Z 390.908, A -75.058, B 83.904, C 170.36, E1 0, E2 0, E3 0, E4 0}
LIN {X 541.887, Y 365.508, Z 391.211, A -75.058, B 83.904, C 170.36, E1 0, E2 0, E3 0, E4 0}
LIN {X 543.962, Y 360.712, Z 391.763, A -75.058, B 83.904, C 170.36, E1 0, E2 0, E3 0, E4 0}
LIN {X 524.149, Y 358.563, Z 391.439, A -75.058, B 83.904, C 170.36, E1 0, E2 0, E3 0, E4 0}
LIN {X 524.615, Y 353.593, Z 391.965, A -75.058, B 83.904, C 170.36, E1 0, E2 0, E3 0, E4 0}
LIN {X 546.13, Y 355.927, Z 392.316, A -75.058, B 83.904, C 170.36, E1 0, E2 0, E3 0, E4 0}
LIN {X 548.298, Y 351.142, Z 392.87, A -75.058, B 83.904, C 170.36, E1 0, E2 0, E3 0, E4 0}
LIN {X 525.318, Y 348.649, Z 392.494, A -75.058, B 83.904, C 170.36, E1 0, E2 0, E3 0, E4 0}
LIN {X 526.299, Y 343.735, Z 393.028, A -75.058, B 83.904, C 170.36, E1 0, E2 0, E3 0, E4 0}
LIN {X 550.466, Y 346.356, Z 393.423, A -75.058, B 83.904, C 170.36, E1 0, E2 0, E3 0, E4 0}
LIN {X 552.634, Y 341.571, Z 393.977, A -75.058, B 83.904, C 170.36, E1 0, E2 0, E3 0, E4 0}
LIN {X 527.195, Y 338.812, Z 393.561, A -75.058, B 83.904, C 170.36, E1 0, E2 0, E3 0, E4 0}
LIN {X 528.308, Y 333.912, Z 394.097, A -75.058, B 83.904, C 170.36, E1 0, E2 0, E3 0, E4 0}
LIN {X 554.802, Y 336.786, Z 394.53, A -75.058, B 83.904, C 170.36, E1 0, E2 0, E3 0, E4 0}
LIN {X 556.971, Y 332, Z 395.084, A -75.058, B 83.904, C 170.36, E1 0, E2 0, E3 0, E4 0}
LIN {X 529.247, Y 328.993, Z 394.631, A -75.058, B 83.904, C 170.36, E1 0, E2 0, E3 0, E4 0}
LIN {X 530.445, Y 324.103, Z 395.168, A -75.058, B 83.904, C 170.36, E1 0, E2 0, E3 0, E4 0}
LIN {X 559.138, Y 327.215, Z 395.637, A -75.058, B 83.904, C 170.36, E1 0, E2 0, E3 0, E4 0}
LIN {X 560.546, Y 322.347, Z 396.178, A -75.058, B 83.904, C 170.36, E1 0, E2 0, E3 0, E4 0}
LIN {X 531.752, Y 319.224, Z 395.708, A -75.058, B 83.904, C 170.36, E1 0, E2 0, E3 0, E4 0}
LIN {X 532.986, Y 314.338, Z 396.246, A -75.058, B 83.904, C 170.36, E1 0, E2 0, E3 0, E4 0}
LIN {X 560.058, Y 317.274, Z 396.688, A -75.058, B 83.904, C 170.36, E1 0, E2 0, E3 0, E4 0}
LIN {X 542.339, Y 310.332, Z 396.917, A -75.058, B 83.904, C 170.36, E1 0, E2 0, E3 0, E4 0}
LIN {X 534.813, Y 309.515, Z 396.793, A -75.058, B 83.904, C 170.36, E1 0, E2 0, E3 0, E4 0}
LIN {X 523.019, Y 367.644, Z 390.471, A -75.058, B 83.904, C 170.36, E1 0, E2 0, E3 0, E4 0}
LIN {X 531.666, Y 319.574, Z 395.669, A -75.058, B 83.904, C 170.36, E1 0, E2 0, E3 0, E4 0}
LIN {X 531.781, Y 318.238, Z 395.81, A -75.058, B 83.904, C 170.36, E1 0, E2 0, E3 0, E4 0}
LIN {X 535.254, Y 308.308, Z 396.93, A -75.058, B 83.904, C 170.36, E1 0, E2 0, E3 0, E4 0}
LIN {X 559.903, Y 315.347, Z 396.883, A -75.058, B 83.904, C 170.36, E1 0, E2 0, E3 0, E4 0}
LIN {X 560.712, Y 323.742, Z 396.039, A -75.058, B 83.904, C 170.36, E1 0, E2 0, E3 0, E4 0}
LIN {X 530.867, Y 392.891, Z 388.082, A -75.058, B 83.904, C 170.36, E1 0, E2 0, E3 0, E4 0}
LIN {X 526.034, Y 392.649, Z 387.974, A -75.058, B 83.904, C 170.36, E1 0, E2 0, E3 0, E4 0}
LIN {X 523.266, Y 391.443, Z 388.022, A -75.058, B 83.904, C 170.36, E1 0, E2 0, E3 0, E4 0}
LIN {X 522.743, Y 391.445, Z 388.007, A -75.058, B 83.904, C 170.36, E1 0, E2 0, E3 0, E4 0}
LIN {X 521.842, Y 391.106, Z 388.017, A -75.058, B 83.904, C 170.36, E1 0, E2 0, E3 0, E4 0}
LIN {X 521.66, Y 390.917, Z 388.032, A -75.058, B 83.904, C 170.36, E1 0, E2 0, E3 0, E4 0}
LIN {X 520.975, Y 389.645, Z 388.144, A -75.058, B 83.904, C 170.36, E1 0, E2 0, E3 0, E4 0}
LIN {X 522.254, Y 371.895, Z 390.011, A -75.058, B 83.904, C 170.36, E1 0, E2 0, E3 0, E4 0}
LIN {X 523.019, Y 367.644, Z 390.471, A -75.058, B 83.904, C 170.36, E1 0, E2 0, E3 0, E4 0}
LIN {X 520.476, Y 388.477, Z 388.251, A -75.058, B 83.904, C 170.36, E1 0, E2 0, E3 0, E4 0}
LIN {X 520.536, Y 388.254, Z 386.09, A -75.058, B 83.904, C 170.36, E1 0, E2 0, E3 0, E4 0}
LIN {X 532.194, Y 389.518, Z 386.28, A -75.058, B 83.904, C 170.36, E1 0, E2 0, E3 0, E4 0}
LIN {X 534.13, Y 384.708, Z 386.83, A -75.058, B 83.904, C 170.36, E1 0, E2 0, E3 0, E4 0}
LIN {X 519.911, Y 383.166, Z 386.597, A -75.058, B 83.904, C 170.36, E1 0, E2 0, E3 0, E4 0}
LIN {X 520.251, Y 378.182, Z 387.121, A -75.058, B 83.904, C 170.36, E1 0, E2 0, E3 0, E4 0}
LIN {X 536.065, Y 379.897, Z 387.379, A -75.058, B 83.904, C 170.36, E1 0, E2 0, E3 0, E4 0}
LIN {X 538.001, Y 375.087, Z 387.929, A -75.058, B 83.904, C 170.36, E1 0, E2 0, E3 0, E4 0}
LIN {X 520.973, Y 373.24, Z 387.651, A -75.058, B 83.904, C 170.36, E1 0, E2 0, E3 0, E4 0}
LIN {X 521.372, Y 368.263, Z 388.175, A -75.058, B 83.904, C 170.36, E1 0, E2 0, E3 0, E4 0}
LIN {X 539.937, Y 370.276, Z 388.479, A -75.058, B 83.904, C 170.36, E1 0, E2 0, E3 0, E4 0}
LIN {X 541.873, Y 365.466, Z 389.028, A -75.058, B 83.904, C 170.36, E1 0, E2 0, E3 0, E4 0}
LIN {X 521.879, Y 363.297, Z 388.702, A -75.058, B 83.904, C 170.36, E1 0, E2 0, E3 0, E4 0}
LIN {X 522.526, Y 358.347, Z 389.23, A -75.058, B 83.904, C 170.36, E1 0, E2 0, E3 0, E4 0}
LIN {X 543.94, Y 360.67, Z 389.58, A -75.058, B 83.904, C 170.36, E1 0, E2 0, E3 0, E4 0}
LIN {X 546.108, Y 355.884, Z 390.134, A -75.058, B 83.904, C 170.36, E1 0, E2 0, E3 0, E4 0}
LIN {X 522.983, Y 353.376, Z 389.756, A -75.058, B 83.904, C 170.36, E1 0, E2 0, E3 0, E4 0}
LIN {X 523.914, Y 348.457, Z 390.289, A -75.058, B 83.904, C 170.36, E1 0, E2 0, E3 0, E4 0}
LIN {X 548.276, Y 351.099, Z 390.687, A -75.058, B 83.904, C 170.36, E1 0, E2 0, E3 0, E4 0}
LIN {X 550.444, Y 346.314, Z 391.241, A -75.058, B 83.904, C 170.36, E1 0, E2 0, E3 0, E4 0}
LIN {X 524.925, Y 343.546, Z 390.824, A -75.058, B 83.904, C 170.36, E1 0, E2 0, E3 0, E4 0}
LIN {X 525.496, Y 338.587, Z 391.351, A -75.058, B 83.904, C 170.36, E1 0, E2 0, E3 0, E4 0}
LIN {X 552.612, Y 341.528, Z 391.794, A -75.058, B 83.904, C 170.36, E1 0, E2 0, E3 0, E4 0}
LIN {X 554.78, Y 336.743, Z 392.348, A -75.058, B 83.904, C 170.36, E1 0, E2 0, E3 0, E4 0}
LIN {X 526.516, Y 333.677, Z 391.886, A -75.058, B 83.904, C 170.36, E1 0, E2 0, E3 0, E4 0}
LIN {X 527.261, Y 328.738, Z 392.416, A -75.058, B 83.904, C 170.36, E1 0, E2 0, E3 0, E4 0}
LIN {X 556.948, Y 331.958, Z 392.901, A -75.058, B 83.904, C 170.36, E1 0, E2 0, E3 0, E4 0}
LIN {X 559.116, Y 327.172, Z 393.455, A -75.058, B 83.904, C 170.36, E1 0, E2 0, E3 0, E4 0}
LIN {X 527.998, Y 323.797, Z 392.946, A -75.058, B 83.904, C 170.36, E1 0, E2 0, E3 0, E4 0}
LIN {X 529.057, Y 318.892, Z 393.481, A -75.058, B 83.904, C 170.36, E1 0, E2 0, E3 0, E4 0}
LIN {X 561.284, Y 322.387, Z 394.008, A -75.058, B 83.904, C 170.36, E1 0, E2 0, E3 0, E4 0}
LIN {X 561.783, Y 317.421, Z 394.534, A -75.058, B 83.904, C 170.36, E1 0, E2 0, E3 0, E4 0}
LIN {X 530.107, Y 313.985, Z 394.017, A -75.058, B 83.904, C 170.36, E1 0, E2 0, E3 0, E4 0}
LIN {X 531.587, Y 309.125, Z 394.559, A -75.058, B 83.904, C 170.36, E1 0, E2 0, E3 0, E4 0}
LIN {X 543.467, Y 310.414, Z 394.753, A -75.058, B 83.904, C 170.36, E1 0, E2 0, E3 0, E4 0}
LIN {X 521.597, Y 366.958, Z 388.316, A -75.058, B 83.904, C 170.36, E1 0, E2 0, E3 0, E4 0}
LIN {X 521.987, Y 362.816, Z 388.754, A -75.058, B 83.904, C 170.36, E1 0, E2 0, E3 0, E4 0}
LIN {X 521.952, Y 362.808, Z 388.754, A -75.058, B 83.904, C 170.36, E1 0, E2 0, E3 0, E4 0}
LIN {X 525.018, Y 342.367, Z 390.948, A -75.058, B 83.904, C 170.36, E1 0, E2 0, E3 0, E4 0}
LIN {X 532.344, Y 306.833, Z 394.816, A -75.058, B 83.904, C 170.36, E1 0, E2 0, E3 0, E4 0}
LIN {X 561.711, Y 315.623, Z 394.718, A -75.058, B 83.904, C 170.36, E1 0, E2 0, E3 0, E4 0}
LIN {X 562.042, Y 320.714, Z 394.202, A -75.058, B 83.904, C 170.36, E1 0, E2 0, E3 0, E4 0}
LIN {X 531.123, Y 392.177, Z 385.976, A -75.058, B 83.904, C 170.36, E1 0, E2 0, E3 0, E4 0}
LIN {X 530.821, Y 392.117, Z 385.974, A -75.058, B 83.904, C 170.36, E1 0, E2 0, E3 0, E4 0}
LIN {X 530.424, Y 391.788, Z 385.997, A -75.058, B 83.904, C 170.36, E1 0, E2 0, E3 0, E4 0}
LIN {X 525.648, Y 390.155, Z 386.034, A -75.058, B 83.904, C 170.36, E1 0, E2 0, E3 0, E4 0}
LIN {X 524.484, Y 390.198, Z 385.998, A -75.058, B 83.904, C 170.36, E1 0, E2 0, E3 0, E4 0}
LIN {X 521.861, Y 391.047, Z 385.838, A -75.058, B 83.904, C 170.36, E1 0, E2 0, E3 0, E4 0}
LIN {X 521.295, Y 390.984, Z 385.829, A -75.058, B 83.904, C 170.36, E1 0, E2 0, E3 0, E4 0}
LIN {X 520.9, Y 390.682, Z 385.849, A -75.058, B 83.904, C 170.36, E1 0, E2 0, E3 0, E4 0}
LIN {X 520.475, Y 389.948, Z 385.913, A -75.058, B 83.904, C 170.36, E1 0, E2 0, E3 0, E4 0}
LIN {X 520.425, Y 389.28, Z 385.981, A -75.058, B 83.904, C 170.36, E1 0, E2 0, E3 0, E4 0}
LIN {X 520.531, Y 388.749, Z 386.038, A -75.058, B 83.904, C 170.36, E1 0, E2 0, E3 0, E4 0}
LIN {X 519.99, Y 384.007, Z 386.513, A -75.058, B 83.904, C 170.36, E1 0, E2 0, E3 0, E4 0}
LIN {X 521.597, Y 366.958, Z 388.316, A -75.058, B 83.904, C 170.36, E1 0, E2 0, E3 0, E4 0}
LIN {X 532.121, Y 389.7, Z 386.259, A -75.058, B 83.904, C 170.36, E1 0, E2 0, E3 0, E4 0}
LIN {X 532.18, Y 389.477, Z 384.098, A -75.058, B 83.904, C 170.36, E1 0, E2 0, E3 0, E4 0}
LIN {X 520.157, Y 388.172, Z 383.901, A -75.058, B 83.904, C 170.36, E1 0, E2 0, E3 0, E4 0}
LIN {X 520.034, Y 383.139, Z 384.417, A -75.058, B 83.904, C 170.36, E1 0, E2 0, E3 0, E4 0}
LIN {X 534.116, Y 384.666, Z 384.647, A -75.058, B 83.904, C 170.36, E1 0, E2 0, E3 0, E4 0}
LIN {X 536.052, Y 379.855, Z 385.197, A -75.058, B 83.904, C 170.36, E1 0, E2 0, E3 0, E4 0}
LIN {X 520.169, Y 378.133, Z 384.938, A -75.058, B 83.904, C 170.36, E1 0, E2 0, E3 0, E4 0}
LIN {X 520.216, Y 373.117, Z 385.456, A -75.058, B 83.904, C 170.36, E1 0, E2 0, E3 0, E4 0}
LIN {X 537.988, Y 375.045, Z 385.747, A -75.058, B 83.904, C 170.36, E1 0, E2 0, E3 0, E4 0}
LIN {X 539.924, Y 370.235, Z 386.297, A -75.058, B 83.904, C 170.36, E1 0, E2 0, E3 0, E4 0}
LIN {X 520.474, Y 368.125, Z 385.979, A -75.058, B 83.904, C 170.36, E1 0, E2 0, E3 0, E4 0}
LIN {X 521.042, Y 363.166, Z 386.506, A -75.058, B 83.904, C 170.36, E1 0, E2 0, E3 0, E4 0}
LIN {X 541.86, Y 365.424, Z 386.846, A -75.058, B 83.904, C 170.36, E1 0, E2 0, E3 0, E4 0}
LIN {X 543.918, Y 360.627, Z 387.398, A -75.058, B 83.904, C 170.36, E1 0, E2 0, E3 0, E4 0}
LIN {X 521.482, Y 358.193, Z 387.031, A -75.058, B 83.904, C 170.36, E1 0, E2 0, E3 0, E4 0}
LIN {X 521.832, Y 353.211, Z 387.555, A -75.058, B 83.904, C 170.36, E1 0, E2 0, E3 0, E4 0}
LIN {X 546.086, Y 355.842, Z 387.951, A -75.058, B 83.904, C 170.36, E1 0, E2 0, E3 0, E4 0}
LIN {X 548.254, Y 351.056, Z 388.505, A -75.058, B 83.904, C 170.36, E1 0, E2 0, E3 0, E4 0}
LIN {X 522.758, Y 348.291, Z 388.088, A -75.058, B 83.904, C 170.36, E1 0, E2 0, E3 0, E4 0}
LIN {X 523.529, Y 343.354, Z 388.619, A -75.058, B 83.904, C 170.36, E1 0, E2 0, E3 0, E4 0}
LIN {X 550.422, Y 346.271, Z 389.058, A -75.058, B 83.904, C 170.36, E1 0, E2 0, E3 0, E4 0}
LIN {X 552.59, Y 341.486, Z 389.612, A -75.058, B 83.904, C 170.36, E1 0, E2 0, E3 0, E4 0}
LIN {X 523.988, Y 338.383, Z 389.144, A -75.058, B 83.904, C 170.36, E1 0, E2 0, E3 0, E4 0}
LIN {X 525.015, Y 333.474, Z 389.679, A -75.058, B 83.904, C 170.36, E1 0, E2 0, E3 0, E4 0}
LIN {X 554.758, Y 336.7, Z 390.165, A -75.058, B 83.904, C 170.36, E1 0, E2 0, E3 0, E4 0}
LIN {X 556.926, Y 331.915, Z 390.719, A -75.058, B 83.904, C 170.36, E1 0, E2 0, E3 0, E4 0}
LIN {X 525.475, Y 328.504, Z 390.205, A -75.058, B 83.904, C 170.36, E1 0, E2 0, E3 0, E4 0}
LIN {X 526.07, Y 323.548, Z 390.732, A -75.058, B 83.904, C 170.36, E1 0, E2 0, E3 0, E4 0}
LIN {X 559.094, Y 327.13, Z 391.272, A -75.058, B 83.904, C 170.36, E1 0, E2 0, E3 0, E4 0}
LIN {X 561.262, Y 322.344, Z 391.826, A -75.058, B 83.904, C 170.36, E1 0, E2 0, E3 0, E4 0}
LIN {X 526.673, Y 318.593, Z 391.26, A -75.058, B 83.904, C 170.36, E1 0, E2 0, E3 0, E4 0}
LIN {X 527.62, Y 313.675, Z 391.794, A -75.058, B 83.904, C 170.36, E1 0, E2 0, E3 0, E4 0}
LIN {X 563.314, Y 317.547, Z 392.377, A -75.058, B 83.904, C 170.36, E1 0, E2 0, E3 0, E4 0}
LIN {X 544.596, Y 310.496, Z 392.589, A -75.058, B 83.904, C 170.36, E1 0, E2 0, E3 0, E4 0}
LIN {X 528.628, Y 308.764, Z 392.328, A -75.058, B 83.904, C 170.36, E1 0, E2 0, E3 0, E4 0}
LIN {X 520.836, Y 366.641, Z 386.142, A -75.058, B 83.904, C 170.36, E1 0, E2 0, E3 0, E4 0}
LIN {X 521.79, Y 355.293, Z 387.339, A -75.058, B 83.904, C 170.36, E1 0, E2 0, E3 0, E4 0}
LIN {X 529.24, Y 305.147, Z 392.718, A -75.058, B 83.904, C 170.36, E1 0, E2 0, E3 0, E4 0}
LIN {X 563.342, Y 315.849, Z 392.553, A -75.058, B 83.904, C 170.36, E1 0, E2 0, E3 0, E4 0}
LIN {X 563.309, Y 317.827, Z 392.348, A -75.058, B 83.904, C 170.36, E1 0, E2 0, E3 0, E4 0}
LIN {X 542.777, Y 363.146, Z 387.107, A -75.058, B 83.904, C 170.36, E1 0, E2 0, E3 0, E4 0}
LIN {X 531.354, Y 391.53, Z 383.863, A -75.058, B 83.904, C 170.36, E1 0, E2 0, E3 0, E4 0}
LIN {X 529.19, Y 390.012, Z 383.96, A -75.058, B 83.904, C 170.36, E1 0, E2 0, E3 0, E4 0}
LIN {X 528.336, Y 389.79, Z 383.96, A -75.058, B 83.904, C 170.36, E1 0, E2 0, E3 0, E4 0}
LIN {X 524.189, Y 390.05, Z 383.819, A -75.058, B 83.904, C 170.36, E1 0, E2 0, E3 0, E4 0}
LIN {X 522.393, Y 390.716, Z 383.7, A -75.058, B 83.904, C 170.36, E1 0, E2 0, E3 0, E4 0}
LIN {X 521.623, Y 390.957, Z 383.654, A -75.058, B 83.904, C 170.36, E1 0, E2 0, E3 0, E4 0}
LIN {X 520.63, Y 390.609, Z 383.663, A -75.058, B 83.904, C 170.36, E1 0, E2 0, E3 0, E4 0}
LIN {X 520.021, Y 389.888, Z 383.721, A -75.058, B 83.904, C 170.36, E1 0, E2 0, E3 0, E4 0}
LIN {X 520.048, Y 376.018, Z 385.152, A -75.058, B 83.904, C 170.36, E1 0, E2 0, E3 0, E4 0}
LIN {X 520.836, Y 366.641, Z 386.142, A -75.058, B 83.904, C 170.36, E1 0, E2 0, E3 0, E4 0}
LIN {X 520.23, Y 388.37, Z 383.883, A -75.058, B 83.904, C 170.36, E1 0, E2 0, E3 0, E4 0}
LIN {X 520.29, Y 388.147, Z 381.721, A -75.058, B 83.904, C 170.36, E1 0, E2 0, E3 0, E4 0}
LIN {X 532.167, Y 389.435, Z 381.915, A -75.058, B 83.904, C 170.36, E1 0, E2 0, E3 0, E4 0}
LIN {X 534.103, Y 384.624, Z 382.465, A -75.058, B 83.904, C 170.36, E1 0, E2 0, E3 0, E4 0}
LIN {X 520.287, Y 383.126, Z 382.239, A -75.058, B 83.904, C 170.36, E1 0, E2 0, E3 0, E4 0}
LIN {X 520.576, Y 378.137, Z 382.762, A -75.058, B 83.904, C 170.36, E1 0, E2 0, E3 0, E4 0}
LIN {X 536.039, Y 379.814, Z 383.015, A -75.058, B 83.904, C 170.36, E1 0, E2 0, E3 0, E4 0}
LIN {X 537.975, Y 375.003, Z 383.564, A -75.058, B 83.904, C 170.36, E1 0, E2 0, E3 0, E4 0}
LIN {X 520.707, Y 373.131, Z 383.282, A -75.058, B 83.904, C 170.36, E1 0, E2 0, E3 0, E4 0}
LIN {X 520.297, Y 368.065, Z 383.794, A -75.058, B 83.904, C 170.36, E1 0, E2 0, E3 0, E4 0}
LIN {X 539.911, Y 370.193, Z 384.114, A -75.058, B 83.904, C 170.36, E1 0, E2 0, E3 0, E4 0}
LIN {X 541.846, Y 365.382, Z 384.664, A -75.058, B 83.904, C 170.36, E1 0, E2 0, E3 0, E4 0}
LIN {X 520.379, Y 363.054, Z 384.313, A -75.058, B 83.904, C 170.36, E1 0, E2 0, E3 0, E4 0}
LIN {X 520.538, Y 358.051, Z 384.833, A -75.058, B 83.904, C 170.36, E1 0, E2 0, E3 0, E4 0}
LIN {X 543.896, Y 360.584, Z 385.215, A -75.058, B 83.904, C 170.36, E1 0, E2 0, E3 0, E4 0}
LIN {X 546.064, Y 355.799, Z 385.769, A -75.058, B 83.904, C 170.36, E1 0, E2 0, E3 0, E4 0}
LIN {X 521.085, Y 353.09, Z 385.36, A -75.058, B 83.904, C 170.36, E1 0, E2 0, E3 0, E4 0}
LIN {X 521.697, Y 348.136, Z 385.888, A -75.058, B 83.904, C 170.36, E1 0, E2 0, E3 0, E4 0}
LIN {X 548.232, Y 351.013, Z 386.322, A -75.058, B 83.904, C 170.36, E1 0, E2 0, E3 0, E4 0}
LIN {X 550.4, Y 346.228, Z 386.876, A -75.058, B 83.904, C 170.36, E1 0, E2 0, E3 0, E4 0}
LIN {X 522.319, Y 343.183, Z 386.417, A -75.058, B 83.904, C 170.36, E1 0, E2 0, E3 0, E4 0}
LIN {X 522.906, Y 338.226, Z 386.944, A -75.058, B 83.904, C 170.36, E1 0, E2 0, E3 0, E4 0}
LIN {X 552.568, Y 341.443, Z 387.429, A -75.058, B 83.904, C 170.36, E1 0, E2 0, E3 0, E4 0}
LIN {X 554.736, Y 336.658, Z 387.983, A -75.058, B 83.904, C 170.36, E1 0, E2 0, E3 0, E4 0}
LIN {X 523.754, Y 333.297, Z 387.476, A -75.058, B 83.904, C 170.36, E1 0, E2 0, E3 0, E4 0}
LIN {X 524.408, Y 328.348, Z 388.005, A -75.058, B 83.904, C 170.36, E1 0, E2 0, E3 0, E4 0}
LIN {X 556.904, Y 331.872, Z 388.536, A -75.058, B 83.904, C 170.36, E1 0, E2 0, E3 0, E4 0}
LIN {X 559.072, Y 327.087, Z 389.09, A -75.058, B 83.904, C 170.36, E1 0, E2 0, E3 0, E4 0}
LIN {X 524.771, Y 323.367, Z 388.529, A -75.058, B 83.904, C 170.36, E1 0, E2 0, E3 0, E4 0}
LIN {X 524.995, Y 318.371, Z 389.051, A -75.058, B 83.904, C 170.36, E1 0, E2 0, E3 0, E4 0}
LIN {X 561.24, Y 322.302, Z 389.643, A -75.058, B 83.904, C 170.36, E1 0, E2 0, E3 0, E4 0}
LIN {X 563.408, Y 317.516, Z 390.196, A -75.058, B 83.904, C 170.36, E1 0, E2 0, E3 0, E4 0}
LIN {X 525.67, Y 313.423, Z 389.58, A -75.058, B 83.904, C 170.36, E1 0, E2 0, E3 0, E4 0}
LIN {X 526.581, Y 308.502, Z 390.113, A -75.058, B 83.904, C 170.36, E1 0, E2 0, E3 0, E4 0}
LIN {X 545.723, Y 310.578, Z 390.426, A -75.058, B 83.904, C 170.36, E1 0, E2 0, E3 0, E4 0}
LIN {X 520.408, Y 366.25, Z 383.984, A -75.058, B 83.904, C 170.36, E1 0, E2 0, E3 0, E4 0}
LIN {X 520.344, Y 364.78, Z 384.134, A -75.058, B 83.904, C 170.36, E1 0, E2 0, E3 0, E4 0}
LIN {X 520.34, Y 364.721, Z 384.14, A -75.058, B 83.904, C 170.36, E1 0, E2 0, E3 0, E4 0}
LIN {X 527.25, Y 303.977, Z 390.598, A -75.058, B 83.904, C 170.36, E1 0, E2 0, E3 0, E4 0}
LIN {X 564.165, Y 315.844, Z 390.39, A -75.058, B 83.904, C 170.36, E1 0, E2 0, E3 0, E4 0}
LIN {X 531.338, Y 391.493, Z 381.68, A -75.058, B 83.904, C 170.36, E1 0, E2 0, E3 0, E4 0}
LIN {X 528.503, Y 389.75, Z 381.782, A -75.058, B 83.904, C 170.36, E1 0, E2 0, E3 0, E4 0}
LIN {X 528.055, Y 389.715, Z 381.773, A -75.058, B 83.904, C 170.36, E1 0, E2 0, E3 0, E4 0}
LIN {X 522.044, Y 390.942, Z 381.481, A -75.058, B 83.904, C 170.36, E1 0, E2 0, E3 0, E4 0}
LIN {X 521.2, Y 390.84, Z 381.468, A -75.058, B 83.904, C 170.36, E1 0, E2 0, E3 0, E4 0}
LIN {X 520.52, Y 390.319, Z 381.503, A -75.058, B 83.904, C 170.36, E1 0, E2 0, E3 0, E4 0}
LIN {X 520.328, Y 389.968, Z 381.534, A -75.058, B 83.904, C 170.36, E1 0, E2 0, E3 0, E4 0}
LIN {X 520.402, Y 374.84, Z 383.097, A -75.058, B 83.904, C 170.36, E1 0, E2 0, E3 0, E4 0}
LIN {X 520.848, Y 372.401, Z 383.361, A -75.058, B 83.904, C 170.36, E1 0, E2 0, E3 0, E4 0}
LIN {X 520.644, Y 371.655, Z 383.433, A -75.058, B 83.904, C 170.36, E1 0, E2 0, E3 0, E4 0}
LIN {X 520.408, Y 366.25, Z 383.984, A -75.058, B 83.904, C 170.36, E1 0, E2 0, E3 0, E4 0}
LIN {X 520.439, Y 388.352, Z 381.704, A -75.058, B 83.904, C 170.36, E1 0, E2 0, E3 0, E4 0}
LIN {X 520.498, Y 388.129, Z 379.543, A -75.058, B 83.904, C 170.36, E1 0, E2 0, E3 0, E4 0}
LIN {X 532.153, Y 389.393, Z 379.733, A -75.058, B 83.904, C 170.36, E1 0, E2 0, E3 0, E4 0}
LIN {X 534.089, Y 384.583, Z 380.283, A -75.058, B 83.904, C 170.36, E1 0, E2 0, E3 0, E4 0}
LIN {X 520.524, Y 383.111, Z 380.061, A -75.058, B 83.904, C 170.36, E1 0, E2 0, E3 0, E4 0}
LIN {X 521.092, Y 378.152, Z 380.588, A -75.058, B 83.904, C 170.36, E1 0, E2 0, E3 0, E4 0}
LIN {X 536.025, Y 379.772, Z 380.832, A -75.058, B 83.904, C 170.36, E1 0, E2 0, E3 0, E4 0}
LIN {X 537.961, Y 374.962, Z 381.382, A -75.058, B 83.904, C 170.36, E1 0, E2 0, E3 0, E4 0}
LIN {X 521.33, Y 373.158, Z 381.11, A -75.058, B 83.904, C 170.36, E1 0, E2 0, E3 0, E4 0}
LIN {X 521.002, Y 368.102, Z 381.623, A -75.058, B 83.904, C 170.36, E1 0, E2 0, E3 0, E4 0}
LIN {X 539.897, Y 370.151, Z 381.932, A -75.058, B 83.904, C 170.36, E1 0, E2 0, E3 0, E4 0}
LIN {X 541.833, Y 365.341, Z 382.481, A -75.058, B 83.904, C 170.36, E1 0, E2 0, E3 0, E4 0}
LIN {X 520.367, Y 363.012, Z 382.131, A -75.058, B 83.904, C 170.36, E1 0, E2 0, E3 0, E4 0}
LIN {X 520.422, Y 357.998, Z 382.65, A -75.058, B 83.904, C 170.36, E1 0, E2 0, E3 0, E4 0}
LIN {X 543.874, Y 360.542, Z 383.033, A -75.058, B 83.904, C 170.36, E1 0, E2 0, E3 0, E4 0}
LIN {X 546.042, Y 355.756, Z 383.586, A -75.058, B 83.904, C 170.36, E1 0, E2 0, E3 0, E4 0}
LIN {X 520.684, Y 353.006, Z 383.172, A -75.058, B 83.904, C 170.36, E1 0, E2 0, E3 0, E4 0}
LIN {X 521.156, Y 348.037, Z 383.698, A -75.058, B 83.904, C 170.36, E1 0, E2 0, E3 0, E4 0}
LIN {X 548.21, Y 350.971, Z 384.14, A -75.058, B 83.904, C 170.36, E1 0, E2 0, E3 0, E4 0}
LIN {X 550.378, Y 346.186, Z 384.693, A -75.058, B 83.904, C 170.36, E1 0, E2 0, E3 0, E4 0}
LIN {X 521.639, Y 343.069, Z 384.224, A -75.058, B 83.904, C 170.36, E1 0, E2 0, E3 0, E4 0}
LIN {X 522.208, Y 338.11, Z 384.751, A -75.058, B 83.904, C 170.36, E1 0, E2 0, E3 0, E4 0}
LIN {X 552.546, Y 341.4, Z 385.247, A -75.058, B 83.904, C 170.36, E1 0, E2 0, E3 0, E4 0}
LIN {X 554.714, Y 336.615, Z 385.8, A -75.058, B 83.904, C 170.36, E1 0, E2 0, E3 0, E4 0}
LIN {X 522.92, Y 333.167, Z 385.281, A -75.058, B 83.904, C 170.36, E1 0, E2 0, E3 0, E4 0}
LIN {X 523.5, Y 328.209, Z 385.808, A -75.058, B 83.904, C 170.36, E1 0, E2 0, E3 0, E4 0}
LIN {X 556.882, Y 331.83, Z 386.354, A -75.058, B 83.904, C 170.36, E1 0, E2 0, E3 0, E4 0}
LIN {X 559.05, Y 327.044, Z 386.907, A -75.058, B 83.904, C 170.36, E1 0, E2 0, E3 0, E4 0}
LIN {X 523.845, Y 323.226, Z 386.332, A -75.058, B 83.904, C 170.36, E1 0, E2 0, E3 0, E4 0}
LIN {X 524.257, Y 318.25, Z 386.857, A -75.058, B 83.904, C 170.36, E1 0, E2 0, E3 0, E4 0}
LIN {X 561.218, Y 322.259, Z 387.461, A -75.058, B 83.904, C 170.36, E1 0, E2 0, E3 0, E4 0}
LIN {X 563.386, Y 317.474, Z 388.014, A -75.058, B 83.904, C 170.36, E1 0, E2 0, E3 0, E4 0}
LIN {X 524.71, Y 313.279, Z 387.382, A -75.058, B 83.904, C 170.36, E1 0, E2 0, E3 0, E4 0}
LIN {X 525.33, Y 308.326, Z 387.91, A -75.058, B 83.904, C 170.36, E1 0, E2 0, E3 0, E4 0}
LIN {X 546.852, Y 310.66, Z 388.262, A -75.058, B 83.904, C 170.36, E1 0, E2 0, E3 0, E4 0}
LIN {X 526.648, Y 303.448, Z 388.45, A -75.058, B 83.904, C 170.36, E1 0, E2 0, E3 0, E4 0}
LIN {X 525.997, Y 303.378, Z 388.439, A -75.058, B 83.904, C 170.36, E1 0, E2 0, E3 0, E4 0}
LIN {X 520.597, Y 366.072, Z 381.821, A -75.058, B 83.904, C 170.36, E1 0, E2 0, E3 0, E4 0}
LIN {X 520.602, Y 355.559, Z 382.906, A -75.058, B 83.904, C 170.36, E1 0, E2 0, E3 0, E4 0}
LIN {X 520.65, Y 353.366, Z 383.134, A -75.058, B 83.904, C 170.36, E1 0, E2 0, E3 0, E4 0}
LIN {X 526.038, Y 303.167, Z 388.462, A -75.058, B 83.904, C 170.36, E1 0, E2 0, E3 0, E4 0}
LIN {X 564.225, Y 315.621, Z 388.228, A -75.058, B 83.904, C 170.36, E1 0, E2 0, E3 0, E4 0}
LIN {X 531.204, Y 391.751, Z 379.464, A -75.058, B 83.904, C 170.36, E1 0, E2 0, E3 0, E4 0}
LIN {X 530.66, Y 391.255, Z 379.5, A -75.058, B 83.904, C 170.36, E1 0, E2 0, E3 0, E4 0}
LIN {X 529.202, Y 389.633, Z 379.627, A -75.058, B 83.904, C 170.36, E1 0, E2 0, E3 0, E4 0}
LIN {X 528.959, Y 389.526, Z 379.631, A -75.058, B 83.904, C 170.36, E1 0, E2 0, E3 0, E4 0}
LIN {X 527.947, Y 389.444, Z 379.612, A -75.058, B 83.904, C 170.36, E1 0, E2 0, E3 0, E4 0}
LIN {X 527.417, Y 389.74, Z 379.567, A -75.058, B 83.904, C 170.36, E1 0, E2 0, E3 0, E4 0}
LIN {X 524.637, Y 390.395, Z 379.423, A -75.058, B 83.904, C 170.36, E1 0, E2 0, E3 0, E4 0}
LIN {X 523.7, Y 391.212, Z 379.313, A -75.058, B 83.904, C 170.36, E1 0, E2 0, E3 0, E4 0}
LIN {X 523.033, Y 391.425, Z 379.272, A -75.058, B 83.904, C 170.36, E1 0, E2 0, E3 0, E4 0}
LIN {X 521.091, Y 390.757, Z 379.288, A -75.058, B 83.904, C 170.36, E1 0, E2 0, E3 0, E4 0}
LIN {X 521.045, Y 390.72, Z 379.29, A -75.058, B 83.904, C 170.36, E1 0, E2 0, E3 0, E4 0}
LIN {X 520.584, Y 389.988, Z 379.353, A -75.058, B 83.904, C 170.36, E1 0, E2 0, E3 0, E4 0}
LIN {X 520.597, Y 366.072, Z 381.821, A -75.058, B 83.904, C 170.36, E1 0, E2 0, E3 0, E4 0}
LIN {X 520.663, Y 388.336, Z 379.526, A -75.058, B 83.904, C 170.36, E1 0, E2 0, E3 0, E4 0}
LIN {X 520.722, Y 388.113, Z 377.364, A -75.058, B 83.904, C 170.36, E1 0, E2 0, E3 0, E4 0}
LIN {X 532.14, Y 389.351, Z 377.551, A -75.058, B 83.904, C 170.36, E1 0, E2 0, E3 0, E4 0}
LIN {X 534.076, Y 384.541, Z 378.1, A -75.058, B 83.904, C 170.36, E1 0, E2 0, E3 0, E4 0}
LIN {X 520.872, Y 383.109, Z 377.885, A -75.058, B 83.904, C 170.36, E1 0, E2 0, E3 0, E4 0}
LIN {X 521.562, Y 378.163, Z 378.414, A -75.058, B 83.904, C 170.36, E1 0, E2 0, E3 0, E4 0}
LIN {X 536.012, Y 379.73, Z 378.65, A -75.058, B 83.904, C 170.36, E1 0, E2 0, E3 0, E4 0}
LIN {X 537.948, Y 374.92, Z 379.2, A -75.058, B 83.904, C 170.36, E1 0, E2 0, E3 0, E4 0}
LIN {X 521.987, Y 373.189, Z 378.939, A -75.058, B 83.904, C 170.36, E1 0, E2 0, E3 0, E4 0}
LIN {X 522.019, Y 368.172, Z 379.457, A -75.058, B 83.904, C 170.36, E1 0, E2 0, E3 0, E4 0}
LIN {X 539.884, Y 370.109, Z 379.749, A -75.058, B 83.904, C 170.36, E1 0, E2 0, E3 0, E4 0}
LIN {X 541.82, Y 365.299, Z 380.299, A -75.058, B 83.904, C 170.36, E1 0, E2 0, E3 0, E4 0}
LIN {X 521.613, Y 363.107, Z 379.969, A -75.058, B 83.904, C 170.36, E1 0, E2 0, E3 0, E4 0}
LIN {X 521.626, Y 358.088, Z 380.487, A -75.058, B 83.904, C 170.36, E1 0, E2 0, E3 0, E4 0}
LIN {X 543.851, Y 360.499, Z 380.85, A -75.058, B 83.904, C 170.36, E1 0, E2 0, E3 0, E4 0}
LIN {X 546.019, Y 355.714, Z 381.404, A -75.058, B 83.904, C 170.36, E1 0, E2 0, E3 0, E4 0}
LIN {X 521.546, Y 353.059, Z 381.004, A -75.058, B 83.904, C 170.36, E1 0, E2 0, E3 0, E4 0}
LIN {X 520.893, Y 347.968, Z 381.511, A -75.058, B 83.904, C 170.36, E1 0, E2 0, E3 0, E4 0}
LIN {X 548.188, Y 350.928, Z 381.957, A -75.058, B 83.904, C 170.36, E1 0, E2 0, E3 0, E4 0}
LIN {X 550.356, Y 346.143, Z 382.511, A -75.058, B 83.904, C 170.36, E1 0, E2 0, E3 0, E4 0}
LIN {X 521.332, Y 342.995, Z 382.036, A -75.058, B 83.904, C 170.36, E1 0, E2 0, E3 0, E4 0}
LIN {X 521.491, Y 337.992, Z 382.557, A -75.058, B 83.904, C 170.36, E1 0, E2 0, E3 0, E4 0}
LIN {X 552.524, Y 341.358, Z 383.064, A -75.058, B 83.904, C 170.36, E1 0, E2 0, E3 0, E4 0}
LIN {X 554.692, Y 336.572, Z 383.618, A -75.058, B 83.904, C 170.36, E1 0, E2 0, E3 0, E4 0}
LIN {X 522.066, Y 333.034, Z 383.084, A -75.058, B 83.904, C 170.36, E1 0, E2 0, E3 0, E4 0}
LIN {X 522.693, Y 328.081, Z 383.613, A -75.058, B 83.904, C 170.36, E1 0, E2 0, E3 0, E4 0}
LIN {X 556.86, Y 331.787, Z 384.171, A -75.058, B 83.904, C 170.36, E1 0, E2 0, E3 0, E4 0}
LIN {X 559.028, Y 327.002, Z 384.725, A -75.058, B 83.904, C 170.36, E1 0, E2 0, E3 0, E4 0}
LIN {X 523.211, Y 323.117, Z 384.139, A -75.058, B 83.904, C 170.36, E1 0, E2 0, E3 0, E4 0}
LIN {X 523.913, Y 318.173, Z 384.669, A -75.058, B 83.904, C 170.36, E1 0, E2 0, E3 0, E4 0}
LIN {X 561.196, Y 322.216, Z 385.278, A -75.058, B 83.904, C 170.36, E1 0, E2 0, E3 0, E4 0}
LIN {X 563.364, Y 317.431, Z 385.832, A -75.058, B 83.904, C 170.36, E1 0, E2 0, E3 0, E4 0}
LIN {X 524.211, Y 313.185, Z 385.192, A -75.058, B 83.904, C 170.36, E1 0, E2 0, E3 0, E4 0}
LIN {X 524.734, Y 308.221, Z 385.718, A -75.058, B 83.904, C 170.36, E1 0, E2 0, E3 0, E4 0}
LIN {X 547.979, Y 310.742, Z 386.098, A -75.058, B 83.904, C 170.36, E1 0, E2 0, E3 0, E4 0}
LIN {X 527.243, Y 303.473, Z 386.277, A -75.058, B 83.904, C 170.36, E1 0, E2 0, E3 0, E4 0}
LIN {X 525.192, Y 303.25, Z 386.244, A -75.058, B 83.904, C 170.36, E1 0, E2 0, E3 0, E4 0}
LIN {X 521.125, Y 365.868, Z 379.671, A -75.058, B 83.904, C 170.36, E1 0, E2 0, E3 0, E4 0}
LIN {X 521.193, Y 360.239, Z 380.253, A -75.058, B 83.904, C 170.36, E1 0, E2 0, E3 0, E4 0}
LIN {X 521.414, Y 359.785, Z 380.306, A -75.058, B 83.904, C 170.36, E1 0, E2 0, E3 0, E4 0}
LIN {X 521.503, Y 352.718, Z 381.038, A -75.058, B 83.904, C 170.36, E1 0, E2 0, E3 0, E4 0}
LIN {X 520.926, Y 351.382, Z 381.16, A -75.058, B 83.904, C 170.36, E1 0, E2 0, E3 0, E4 0}
LIN {X 525.257, Y 302.555, Z 386.317, A -75.058, B 83.904, C 170.36, E1 0, E2 0, E3 0, E4 0}
LIN {X 564.285, Y 315.398, Z 386.067, A -75.058, B 83.904, C 170.36, E1 0, E2 0, E3 0, E4 0}
LIN {X 530.932, Y 392.353, Z 377.208, A -75.058, B 83.904, C 170.36, E1 0, E2 0, E3 0, E4 0}
LIN {X 530.814, Y 392.328, Z 377.207, A -75.058, B 83.904, C 170.36, E1 0, E2 0, E3 0, E4 0}
LIN {X 527.287, Y 392.125, Z 377.131, A -75.058, B 83.904, C 170.36, E1 0, E2 0, E3 0, E4 0}
LIN {X 523.977, Y 391.612, Z 377.093, A -75.058, B 83.904, C 170.36, E1 0, E2 0, E3 0, E4 0}
LIN {X 521.51, Y 390.186, Z 377.172, A -75.058, B 83.904, C 170.36, E1 0, E2 0, E3 0, E4 0}
LIN {X 520.848, Y 388.846, Z 377.292, A -75.058, B 83.904, C 170.36, E1 0, E2 0, E3 0, E4 0}
LIN {X 521.125, Y 365.868, Z 379.671, A -75.058, B 83.904, C 170.36, E1 0, E2 0, E3 0, E4 0}
LIN {X 520.982, Y 388.33, Z 377.349, A -75.058, B 83.904, C 170.36, E1 0, E2 0, E3 0, E4 0}
LIN {X 521.042, Y 388.107, Z 375.187, A -75.058, B 83.904, C 170.36, E1 0, E2 0, E3 0, E4 0}
LIN {X 532.126, Y 389.31, Z 375.369, A -75.058, B 83.904, C 170.36, E1 0, E2 0, E3 0, E4 0}
LIN {X 534.062, Y 384.499, Z 375.918, A -75.058, B 83.904, C 170.36, E1 0, E2 0, E3 0, E4 0}
LIN {X 521.266, Y 383.111, Z 375.709, A -75.058, B 83.904, C 170.36, E1 0, E2 0, E3 0, E4 0}
LIN {X 522.074, Y 378.178, Z 376.24, A -75.058, B 83.904, C 170.36, E1 0, E2 0, E3 0, E4 0}
LIN {X 535.998, Y 379.689, Z 376.468, A -75.058, B 83.904, C 170.36, E1 0, E2 0, E3 0, E4 0}
LIN {X 537.934, Y 374.878, Z 377.017, A -75.058, B 83.904, C 170.36, E1 0, E2 0, E3 0, E4 0}
LIN {X 522.45, Y 373.199, Z 376.764, A -75.058, B 83.904, C 170.36, E1 0, E2 0, E3 0, E4 0}
LIN {X 522.704, Y 368.206, Z 377.286, A -75.058, B 83.904, C 170.36, E1 0, E2 0, E3 0, E4 0}
LIN {X 539.87, Y 370.068, Z 377.567, A -75.058, B 83.904, C 170.36, E1 0, E2 0, E3 0, E4 0}
LIN {X 541.806, Y 365.257, Z 378.117, A -75.058, B 83.904, C 170.36, E1 0, E2 0, E3 0, E4 0}
LIN {X 523.311, Y 363.251, Z 377.815, A -75.058, B 83.904, C 170.36, E1 0, E2 0, E3 0, E4 0}
LIN {X 522.71, Y 358.166, Z 378.323, A -75.058, B 83.904, C 170.36, E1 0, E2 0, E3 0, E4 0}
LIN {X 543.829, Y 360.456, Z 378.668, A -75.058, B 83.904, C 170.36, E1 0, E2 0, E3 0, E4 0}
LIN {X 545.997, Y 355.671, Z 379.221, A -75.058, B 83.904, C 170.36, E1 0, E2 0, E3 0, E4 0}
LIN {X 522.598, Y 353.133, Z 378.839, A -75.058, B 83.904, C 170.36, E1 0, E2 0, E3 0, E4 0}
LIN {X 522.173, Y 348.066, Z 379.35, A -75.058, B 83.904, C 170.36, E1 0, E2 0, E3 0, E4 0}
LIN {X 548.165, Y 350.885, Z 379.775, A -75.058, B 83.904, C 170.36, E1 0, E2 0, E3 0, E4 0}
LIN {X 550.333, Y 346.1, Z 380.328, A -75.058, B 83.904, C 170.36, E1 0, E2 0, E3 0, E4 0}
LIN {X 521.976, Y 343.025, Z 379.865, A -75.058, B 83.904, C 170.36, E1 0, E2 0, E3 0, E4 0}
LIN {X 521.71, Y 337.975, Z 380.379, A -75.058, B 83.904, C 170.36, E1 0, E2 0, E3 0, E4 0}
LIN {X 552.501, Y 341.315, Z 380.882, A -75.058, B 83.904, C 170.36, E1 0, E2 0, E3 0, E4 0}
LIN {X 554.669, Y 336.53, Z 381.435, A -75.058, B 83.904, C 170.36, E1 0, E2 0, E3 0, E4 0}
LIN {X 522.212, Y 333.009, Z 380.905, A -75.058, B 83.904, C 170.36, E1 0, E2 0, E3 0, E4 0}
LIN {X 522.253, Y 327.993, Z 381.423, A -75.058, B 83.904, C 170.36, E1 0, E2 0, E3 0, E4 0}
LIN {X 556.837, Y 331.744, Z 381.989, A -75.058, B 83.904, C 170.36, E1 0, E2 0, E3 0, E4 0}
LIN {X 559.005, Y 326.959, Z 382.542, A -75.058, B 83.904, C 170.36, E1 0, E2 0, E3 0, E4 0}
LIN {X 522.714, Y 323.023, Z 381.949, A -75.058, B 83.904, C 170.36, E1 0, E2 0, E3 0, E4 0}
LIN {X 523.416, Y 318.079, Z 382.479, A -75.058, B 83.904, C 170.36, E1 0, E2 0, E3 0, E4 0}
LIN {X 561.173, Y 322.174, Z 383.096, A -75.058, B 83.904, C 170.36, E1 0, E2 0, E3 0, E4 0}
LIN {X 563.341, Y 317.388, Z 383.649, A -75.058, B 83.904, C 170.36, E1 0, E2 0, E3 0, E4 0}
LIN {X 523.959, Y 313.117, Z 383.005, A -75.058, B 83.904, C 170.36, E1 0, E2 0, E3 0, E4 0}
LIN {X 524.423, Y 308.147, Z 383.531, A -75.058, B 83.904, C 170.36, E1 0, E2 0, E3 0, E4 0}
LIN {X 549.107, Y 310.824, Z 383.934, A -75.058, B 83.904, C 170.36, E1 0, E2 0, E3 0, E4 0}
LIN {X 527.836, Y 303.497, Z 384.105, A -75.058, B 83.904, C 170.36, E1 0, E2 0, E3 0, E4 0}
LIN {X 524.771, Y 303.164, Z 384.055, A -75.058, B 83.904, C 170.36, E1 0, E2 0, E3 0, E4 0}
LIN {X 523.159, Y 365.953, Z 377.531, A -75.058, B 83.904, C 170.36, E1 0, E2 0, E3 0, E4 0}
LIN {X 523.341, Y 363.953, Z 377.743, A -75.058, B 83.904, C 170.36, E1 0, E2 0, E3 0, E4 0}
LIN {X 523.116, Y 360.476, Z 378.096, A -75.058, B 83.904, C 170.36, E1 0, E2 0, E3 0, E4 0}
LIN {X 523.192, Y 360.262, Z 378.12, A -75.058, B 83.904, C 170.36, E1 0, E2 0, E3 0, E4 0}
LIN {X 523.051, Y 359.956, Z 378.147, A -75.058, B 83.904, C 170.36, E1 0, E2 0, E3 0, E4 0}
LIN {X 522.643, Y 352.859, Z 378.868, A -75.058, B 83.904, C 170.36, E1 0, E2 0, E3 0, E4 0}
LIN {X 522.498, Y 351.968, Z 378.956, A -75.058, B 83.904, C 170.36, E1 0, E2 0, E3 0, E4 0}
LIN {X 522.326, Y 351.675, Z 378.982, A -75.058, B 83.904, C 170.36, E1 0, E2 0, E3 0, E4 0}
LIN {X 522.122, Y 350.456, Z 379.102, A -75.058, B 83.904, C 170.36, E1 0, E2 0, E3 0, E4 0}
LIN {X 522.102, Y 350.414, Z 379.106, A -75.058, B 83.904, C 170.36, E1 0, E2 0, E3 0, E4 0}
LIN {X 522.11, Y 348.265, Z 379.328, A -75.058, B 83.904, C 170.36, E1 0, E2 0, E3 0, E4 0}
LIN {X 522.185, Y 348.259, Z 379.331, A -75.058, B 83.904, C 170.36, E1 0, E2 0, E3 0, E4 0}
LIN {X 522.151, Y 347.715, Z 379.386, A -75.058, B 83.904, C 170.36, E1 0, E2 0, E3 0, E4 0}
LIN {X 522.032, Y 347.699, Z 379.384, A -75.058, B 83.904, C 170.36, E1 0, E2 0, E3 0, E4 0}
LIN {X 522.372, Y 329.673, Z 381.253, A -75.058, B 83.904, C 170.36, E1 0, E2 0, E3 0, E4 0}
LIN {X 522.284, Y 329.249, Z 381.295, A -75.058, B 83.904, C 170.36, E1 0, E2 0, E3 0, E4 0}
LIN {X 524.828, Y 302.106, Z 384.165, A -75.058, B 83.904, C 170.36, E1 0, E2 0, E3 0, E4 0}
LIN {X 564.344, Y 315.175, Z 383.905, A -75.058, B 83.904, C 170.36, E1 0, E2 0, E3 0, E4 0}
LIN {X 530.873, Y 392.424, Z 375.013, A -75.058, B 83.904, C 170.36, E1 0, E2 0, E3 0, E4 0}
LIN {X 530.647, Y 392.462, Z 375.002, A -75.058, B 83.904, C 170.36, E1 0, E2 0, E3 0, E4 0}
LIN {X 526.064, Y 392.041, Z 374.92, A -75.058, B 83.904, C 170.36, E1 0, E2 0, E3 0, E4 0}
LIN {X 521.415, Y 389.657, Z 375.038, A -75.058, B 83.904, C 170.36, E1 0, E2 0, E3 0, E4 0}
LIN {X 521.097, Y 388.607, Z 375.137, A -75.058, B 83.904, C 170.36, E1 0, E2 0, E3 0, E4 0}
LIN {X 523.159, Y 365.953, Z 377.531, A -75.058, B 83.904, C 170.36, E1 0, E2 0, E3 0, E4 0}
LIN {X 521.576, Y 388.354, Z 375.176, A -75.058, B 83.904, C 170.36, E1 0, E2 0, E3 0, E4 0}
LIN {X 521.636, Y 388.131, Z 373.015, A -75.058, B 83.904, C 170.36, E1 0, E2 0, E3 0, E4 0}
LIN {X 532.113, Y 389.268, Z 373.186, A -75.058, B 83.904, C 170.36, E1 0, E2 0, E3 0, E4 0}
LIN {X 534.049, Y 384.457, Z 373.736, A -75.058, B 83.904, C 170.36, E1 0, E2 0, E3 0, E4 0}
LIN {X 521.787, Y 383.127, Z 373.535, A -75.058, B 83.904, C 170.36, E1 0, E2 0, E3 0, E4 0}
LIN {X 522.875, Y 378.225, Z 374.071, A -75.058, B 83.904, C 170.36, E1 0, E2 0, E3 0, E4 0}
LIN {X 535.985, Y 379.647, Z 374.285, A -75.058, B 83.904, C 170.36, E1 0, E2 0, E3 0, E4 0}
LIN {X 537.921, Y 374.836, Z 374.835, A -75.058, B 83.904, C 170.36, E1 0, E2 0, E3 0, E4 0}
LIN {X 522.974, Y 373.215, Z 374.591, A -75.058, B 83.904, C 170.36, E1 0, E2 0, E3 0, E4 0}
LIN {X 523.309, Y 368.231, Z 375.114, A -75.058, B 83.904, C 170.36, E1 0, E2 0, E3 0, E4 0}
LIN {X 539.857, Y 370.026, Z 375.385, A -75.058, B 83.904, C 170.36, E1 0, E2 0, E3 0, E4 0}
LIN {X 541.793, Y 365.215, Z 375.935, A -75.058, B 83.904, C 170.36, E1 0, E2 0, E3 0, E4 0}
LIN {X 523.874, Y 363.272, Z 375.642, A -75.058, B 83.904, C 170.36, E1 0, E2 0, E3 0, E4 0}
LIN {X 523.831, Y 358.247, Z 376.159, A -75.058, B 83.904, C 170.36, E1 0, E2 0, E3 0, E4 0}
LIN {X 543.807, Y 360.414, Z 376.486, A -75.058, B 83.904, C 170.36, E1 0, E2 0, E3 0, E4 0}
LIN {X 545.975, Y 355.628, Z 377.039, A -75.058, B 83.904, C 170.36, E1 0, E2 0, E3 0, E4 0}
LIN {X 523.734, Y 353.216, Z 376.675, A -75.058, B 83.904, C 170.36, E1 0, E2 0, E3 0, E4 0}
LIN {X 523.129, Y 348.13, Z 377.183, A -75.058, B 83.904, C 170.36, E1 0, E2 0, E3 0, E4 0}
LIN {X 548.143, Y 350.843, Z 377.592, A -75.058, B 83.904, C 170.36, E1 0, E2 0, E3 0, E4 0}
LIN {X 550.311, Y 346.058, Z 378.146, A -75.058, B 83.904, C 170.36, E1 0, E2 0, E3 0, E4 0}
LIN {X 523.277, Y 343.125, Z 377.704, A -75.058, B 83.904, C 170.36, E1 0, E2 0, E3 0, E4 0}
LIN {X 523.186, Y 338.095, Z 378.22, A -75.058, B 83.904, C 170.36, E1 0, E2 0, E3 0, E4 0}
LIN {X 552.479, Y 341.272, Z 378.699, A -75.058, B 83.904, C 170.36, E1 0, E2 0, E3 0, E4 0}
LIN {X 554.647, Y 336.487, Z 379.253, A -75.058, B 83.904, C 170.36, E1 0, E2 0, E3 0, E4 0}
LIN {X 523.664, Y 333.127, Z 378.746, A -75.058, B 83.904, C 170.36, E1 0, E2 0, E3 0, E4 0}
LIN {X 523.343, Y 328.071, Z 379.259, A -75.058, B 83.904, C 170.36, E1 0, E2 0, E3 0, E4 0}
LIN {X 556.815, Y 331.702, Z 379.806, A -75.058, B 83.904, C 170.36, E1 0, E2 0, E3 0, E4 0}
LIN {X 558.983, Y 326.916, Z 380.36, A -75.058, B 83.904, C 170.36, E1 0, E2 0, E3 0, E4 0}
LIN {X 522.892, Y 323.002, Z 379.77, A -75.058, B 83.904, C 170.36, E1 0, E2 0, E3 0, E4 0}
LIN {X 523.245, Y 318.02, Z 380.293, A -75.058, B 83.904, C 170.36, E1 0, E2 0, E3 0, E4 0}
LIN {X 561.151, Y 322.131, Z 380.913, A -75.058, B 83.904, C 170.36, E1 0, E2 0, E3 0, E4 0}
LIN {X 563.319, Y 317.346, Z 381.467, A -75.058, B 83.904, C 170.36, E1 0, E2 0, E3 0, E4 0}
LIN {X 523.765, Y 313.056, Z 380.82, A -75.058, B 83.904, C 170.36, E1 0, E2 0, E3 0, E4 0}
LIN {X 524.116, Y 308.073, Z 381.344, A -75.058, B 83.904, C 170.36, E1 0, E2 0, E3 0, E4 0}
LIN {X 550.236, Y 310.906, Z 381.771, A -75.058, B 83.904, C 170.36, E1 0, E2 0, E3 0, E4 0}
LIN {X 528.431, Y 303.521, Z 381.932, A -75.058, B 83.904, C 170.36, E1 0, E2 0, E3 0, E4 0}
LIN {X 524.507, Y 303.095, Z 381.868, A -75.058, B 83.904, C 170.36, E1 0, E2 0, E3 0, E4 0}
LIN {X 523.674, Y 365.781, Z 375.377, A -75.058, B 83.904, C 170.36, E1 0, E2 0, E3 0, E4 0}
LIN {X 523.784, Y 364.599, Z 375.502, A -75.058, B 83.904, C 170.36, E1 0, E2 0, E3 0, E4 0}
LIN {X 523.157, Y 338.44, Z 378.184, A -75.058, B 83.904, C 170.36, E1 0, E2 0, E3 0, E4 0}
LIN {X 523.838, Y 335.305, Z 378.526, A -75.058, B 83.904, C 170.36, E1 0, E2 0, E3 0, E4 0}
LIN {X 522.845, Y 325.324, Z 379.529, A -75.058, B 83.904, C 170.36, E1 0, E2 0, E3 0, E4 0}
LIN {X 522.815, Y 325.206, Z 379.54, A -75.058, B 83.904, C 170.36, E1 0, E2 0, E3 0, E4 0}
LIN {X 524.586, Y 301.744, Z 382.01, A -75.058, B 83.904, C 170.36, E1 0, E2 0, E3 0, E4 0}
LIN {X 564.404, Y 314.952, Z 381.743, A -75.058, B 83.904, C 170.36, E1 0, E2 0, E3 0, E4 0}
LIN {X 530.888, Y 392.312, Z 372.838, A -75.058, B 83.904, C 170.36, E1 0, E2 0, E3 0, E4 0}
LIN {X 530.763, Y 392.326, Z 372.833, A -75.058, B 83.904, C 170.36, E1 0, E2 0, E3 0, E4 0}
LIN {X 530.283, Y 392.443, Z 372.808, A -75.058, B 83.904, C 170.36, E1 0, E2 0, E3 0, E4 0}
LIN {X 521.924, Y 390.369, Z 372.792, A -75.058, B 83.904, C 170.36, E1 0, E2 0, E3 0, E4 0}
LIN {X 521.573, Y 389.717, Z 372.85, A -75.058, B 83.904, C 170.36, E1 0, E2 0, E3 0, E4 0}
LIN {X 521.616, Y 388.191, Z 373.008, A -75.058, B 83.904, C 170.36, E1 0, E2 0, E3 0, E4 0}
LIN {X 521.631, Y 388.162, Z 373.012, A -75.058, B 83.904, C 170.36, E1 0, E2 0, E3 0, E4 0}
LIN {X 521.741, Y 385.435, Z 373.296, A -75.058, B 83.904, C 170.36, E1 0, E2 0, E3 0, E4 0}
LIN {X 521.814, Y 384.578, Z 373.386, A -75.058, B 83.904, C 170.36, E1 0, E2 0, E3 0, E4 0}
LIN {X 521.748, Y 384.505, Z 373.392, A -75.058, B 83.904, C 170.36, E1 0, E2 0, E3 0, E4 0}
LIN {X 521.664, Y 384.044, Z 373.437, A -75.058, B 83.904, C 170.36, E1 0, E2 0, E3 0, E4 0}
LIN {X 522.144, Y 382.228, Z 373.638, A -75.058, B 83.904, C 170.36, E1 0, E2 0, E3 0, E4 0}
LIN {X 523.674, Y 365.781, Z 375.377, A -75.058, B 83.904, C 170.36, E1 0, E2 0, E3 0, E4 0}
LIN {X 522.347, Y 388.398, Z 373.007, A -75.058, B 83.904, C 170.36, E1 0, E2 0, E3 0, E4 0}
LIN {X 522.407, Y 388.175, Z 370.845, A -75.058, B 83.904, C 170.36, E1 0, E2 0, E3 0, E4 0}
LIN {X 532.1, Y 389.226, Z 371.004, A -75.058, B 83.904, C 170.36, E1 0, E2 0, E3 0, E4 0}
LIN {X 534.035, Y 384.416, Z 371.553, A -75.058, B 83.904, C 170.36, E1 0, E2 0, E3 0, E4 0}
LIN {X 523.014, Y 383.22, Z 371.373, A -75.058, B 83.904, C 170.36, E1 0, E2 0, E3 0, E4 0}
LIN {X 523.645, Y 378.268, Z 371.902, A -75.058, B 83.904, C 170.36, E1 0, E2 0, E3 0, E4 0}
LIN {X 535.971, Y 379.605, Z 372.103, A -75.058, B 83.904, C 170.36, E1 0, E2 0, E3 0, E4 0}
LIN {X 537.907, Y 374.795, Z 372.653, A -75.058, B 83.904, C 170.36, E1 0, E2 0, E3 0, E4 0}
LIN {X 523.649, Y 373.248, Z 372.42, A -75.058, B 83.904, C 170.36, E1 0, E2 0, E3 0, E4 0}
LIN {X 523.996, Y 368.265, Z 372.943, A -75.058, B 83.904, C 170.36, E1 0, E2 0, E3 0, E4 0}
LIN {X 539.843, Y 369.984, Z 373.202, A -75.058, B 83.904, C 170.36, E1 0, E2 0, E3 0, E4 0}
LIN {X 541.779, Y 365.174, Z 373.752, A -75.058, B 83.904, C 170.36, E1 0, E2 0, E3 0, E4 0}
LIN {X 524.489, Y 363.298, Z 373.469, A -75.058, B 83.904, C 170.36, E1 0, E2 0, E3 0, E4 0}
LIN {X 524.573, Y 358.287, Z 373.989, A -75.058, B 83.904, C 170.36, E1 0, E2 0, E3 0, E4 0}
LIN {X 543.785, Y 360.371, Z 374.303, A -75.058, B 83.904, C 170.36, E1 0, E2 0, E3 0, E4 0}
LIN {X 545.953, Y 355.585, Z 374.856, A -75.058, B 83.904, C 170.36, E1 0, E2 0, E3 0, E4 0}
LIN {X 524.388, Y 353.247, Z 374.504, A -75.058, B 83.904, C 170.36, E1 0, E2 0, E3 0, E4 0}
LIN {X 524.294, Y 348.216, Z 375.021, A -75.058, B 83.904, C 170.36, E1 0, E2 0, E3 0, E4 0}
LIN {X 548.121, Y 350.8, Z 375.41, A -75.058, B 83.904, C 170.36, E1 0, E2 0, E3 0, E4 0}
LIN {X 550.289, Y 346.015, Z 375.963, A -75.058, B 83.904, C 170.36, E1 0, E2 0, E3 0, E4 0}
LIN {X 524.433, Y 343.211, Z 375.541, A -75.058, B 83.904, C 170.36, E1 0, E2 0, E3 0, E4 0}
LIN {X 524.906, Y 338.241, Z 376.066, A -75.058, B 83.904, C 170.36, E1 0, E2 0, E3 0, E4 0}
LIN {X 552.457, Y 341.23, Z 376.517, A -75.058, B 83.904, C 170.36, E1 0, E2 0, E3 0, E4 0}
LIN {X 554.625, Y 336.444, Z 377.07, A -75.058, B 83.904, C 170.36, E1 0, E2 0, E3 0, E4 0}
LIN {X 524.833, Y 333.213, Z 376.583, A -75.058, B 83.904, C 170.36, E1 0, E2 0, E3 0, E4 0}
LIN {X 524.574, Y 328.164, Z 377.097, A -75.058, B 83.904, C 170.36, E1 0, E2 0, E3 0, E4 0}
LIN {X 556.793, Y 331.659, Z 377.624, A -75.058, B 83.904, C 170.36, E1 0, E2 0, E3 0, E4 0}
LIN {X 558.961, Y 326.874, Z 378.177, A -75.058, B 83.904, C 170.36, E1 0, E2 0, E3 0, E4 0}
LIN {X 524.166, Y 323.1, Z 377.609, A -75.058, B 83.904, C 170.36, E1 0, E2 0, E3 0, E4 0}
LIN {X 523.669, Y 318.025, Z 378.118, A -75.058, B 83.904, C 170.36, E1 0, E2 0, E3 0, E4 0}
LIN {X 561.129, Y 322.088, Z 378.731, A -75.058, B 83.904, C 170.36, E1 0, E2 0, E3 0, E4 0}
LIN {X 563.297, Y 317.303, Z 379.284, A -75.058, B 83.904, C 170.36, E1 0, E2 0, E3 0, E4 0}
LIN {X 524.08, Y 313.05, Z 378.643, A -75.058, B 83.904, C 170.36, E1 0, E2 0, E3 0, E4 0}
LIN {X 524.33, Y 308.056, Z 379.165, A -75.058, B 83.904, C 170.36, E1 0, E2 0, E3 0, E4 0}
LIN {X 551.363, Y 310.988, Z 379.607, A -75.058, B 83.904, C 170.36, E1 0, E2 0, E3 0, E4 0}
LIN {X 529.027, Y 303.545, Z 379.76, A -75.058, B 83.904, C 170.36, E1 0, E2 0, E3 0, E4 0}
LIN {X 524.753, Y 303.082, Z 379.69, A -75.058, B 83.904, C 170.36, E1 0, E2 0, E3 0, E4 0}
LIN {X 523.901, Y 365.214, Z 373.256, A -75.058, B 83.904, C 170.36, E1 0, E2 0, E3 0, E4 0}
LIN {X 524.256, Y 309.367, Z 379.028, A -75.058, B 83.904, C 170.36, E1 0, E2 0, E3 0, E4 0}
LIN {X 524.84, Y 301.61, Z 379.845, A -75.058, B 83.904, C 170.36, E1 0, E2 0, E3 0, E4 0}
LIN {X 564.463, Y 314.729, Z 379.582, A -75.058, B 83.904, C 170.36, E1 0, E2 0, E3 0, E4 0}
LIN {X 530.935, Y 392.121, Z 370.673, A -75.058, B 83.904, C 170.36, E1 0, E2 0, E3 0, E4 0}
LIN {X 530.613, Y 392.122, Z 370.664, A -75.058, B 83.904, C 170.36, E1 0, E2 0, E3 0, E4 0}
LIN {X 530.57, Y 392.132, Z 370.662, A -75.058, B 83.904, C 170.36, E1 0, E2 0, E3 0, E4 0}
LIN {X 521.961, Y 390.657, Z 370.577, A -75.058, B 83.904, C 170.36, E1 0, E2 0, E3 0, E4 0}
LIN {X 521.748, Y 390.494, Z 370.588, A -75.058, B 83.904, C 170.36, E1 0, E2 0, E3 0, E4 0}
LIN {X 521.492, Y 390.089, Z 370.623, A -75.058, B 83.904, C 170.36, E1 0, E2 0, E3 0, E4 0}
LIN {X 521.49, Y 390.069, Z 370.625, A -75.058, B 83.904, C 170.36, E1 0, E2 0, E3 0, E4 0}
LIN {X 522.983, Y 386.893, Z 370.993, A -75.058, B 83.904, C 170.36, E1 0, E2 0, E3 0, E4 0}
LIN {X 523.014, Y 383.22, Z 371.373, A -75.058, B 83.904, C 170.36, E1 0, E2 0, E3 0, E4 0}
LIN {X 523.801, Y 380.939, Z 371.63, A -75.058, B 83.904, C 170.36, E1 0, E2 0, E3 0, E4 0}
LIN {X 523.901, Y 365.214, Z 373.256, A -75.058, B 83.904, C 170.36, E1 0, E2 0, E3 0, E4 0}
LIN {X 522.868, Y 388.414, Z 370.833, A -75.058, B 83.904, C 170.36, E1 0, E2 0, E3 0, E4 0}
LIN {X 522.927, Y 388.191, Z 368.672, A -75.058, B 83.904, C 170.36, E1 0, E2 0, E3 0, E4 0}
LIN {X 532.086, Y 389.184, Z 368.821, A -75.058, B 83.904, C 170.36, E1 0, E2 0, E3 0, E4 0}
LIN {X 534.022, Y 384.374, Z 369.371, A -75.058, B 83.904, C 170.36, E1 0, E2 0, E3 0, E4 0}
LIN {X 524.249, Y 383.314, Z 369.211, A -75.058, B 83.904, C 170.36, E1 0, E2 0, E3 0, E4 0}
LIN {X 524.273, Y 378.296, Z 369.73, A -75.058, B 83.904, C 170.36, E1 0, E2 0, E3 0, E4 0}
LIN {X 535.958, Y 379.563, Z 369.921, A -75.058, B 83.904, C 170.36, E1 0, E2 0, E3 0, E4 0}
LIN {X 537.894, Y 374.753, Z 370.47, A -75.058, B 83.904, C 170.36, E1 0, E2 0, E3 0, E4 0}
LIN {X 524.571, Y 373.308, Z 370.253, A -75.058, B 83.904, C 170.36, E1 0, E2 0, E3 0, E4 0}
LIN {X 524.834, Y 368.316, Z 370.775, A -75.058, B 83.904, C 170.36, E1 0, E2 0, E3 0, E4 0}
LIN {X 539.83, Y 369.943, Z 371.02, A -75.058, B 83.904, C 170.36, E1 0, E2 0, E3 0, E4 0}
LIN {X 541.766, Y 365.132, Z 371.57, A -75.058, B 83.904, C 170.36, E1 0, E2 0, E3 0, E4 0}
LIN {X 525.325, Y 363.349, Z 371.301, A -75.058, B 83.904, C 170.36, E1 0, E2 0, E3 0, E4 0}
LIN {X 525.602, Y 358.358, Z 371.823, A -75.058, B 83.904, C 170.36, E1 0, E2 0, E3 0, E4 0}
LIN {X 543.763, Y 360.328, Z 372.12, A -75.058, B 83.904, C 170.36, E1 0, E2 0, E3 0, E4 0}
LIN {X 545.931, Y 355.543, Z 372.674, A -75.058, B 83.904, C 170.36, E1 0, E2 0, E3 0, E4 0}
LIN {X 525.379, Y 353.314, Z 372.338, A -75.058, B 83.904, C 170.36, E1 0, E2 0, E3 0, E4 0}
LIN {X 525.653, Y 348.323, Z 372.86, A -75.058, B 83.904, C 170.36, E1 0, E2 0, E3 0, E4 0}
LIN {X 548.099, Y 350.758, Z 373.227, A -75.058, B 83.904, C 170.36, E1 0, E2 0, E3 0, E4 0}
LIN {X 550.267, Y 345.972, Z 373.781, A -75.058, B 83.904, C 170.36, E1 0, E2 0, E3 0, E4 0}
LIN {X 525.92, Y 343.332, Z 373.383, A -75.058, B 83.904, C 170.36, E1 0, E2 0, E3 0, E4 0}
LIN {X 525.991, Y 338.319, Z 373.902, A -75.058, B 83.904, C 170.36, E1 0, E2 0, E3 0, E4 0}
LIN {X 552.435, Y 341.187, Z 374.334, A -75.058, B 83.904, C 170.36, E1 0, E2 0, E3 0, E4 0}
LIN {X 554.603, Y 336.402, Z 374.888, A -75.058, B 83.904, C 170.36, E1 0, E2 0, E3 0, E4 0}
LIN {X 525.934, Y 333.292, Z 374.419, A -75.058, B 83.904, C 170.36, E1 0, E2 0, E3 0, E4 0}
LIN {X 525.975, Y 328.276, Z 374.938, A -75.058, B 83.904, C 170.36, E1 0, E2 0, E3 0, E4 0}
LIN {X 556.771, Y 331.616, Z 375.441, A -75.058, B 83.904, C 170.36, E1 0, E2 0, E3 0, E4 0}
LIN {X 558.939, Y 326.831, Z 375.995, A -75.058, B 83.904, C 170.36, E1 0, E2 0, E3 0, E4 0}
LIN {X 526.075, Y 323.267, Z 375.458, A -75.058, B 83.904, C 170.36, E1 0, E2 0, E3 0, E4 0}
LIN {X 525.182, Y 318.149, Z 375.961, A -75.058, B 83.904, C 170.36, E1 0, E2 0, E3 0, E4 0}
LIN {X 561.107, Y 322.046, Z 376.548, A -75.058, B 83.904, C 170.36, E1 0, E2 0, E3 0, E4 0}
LIN {X 563.275, Y 317.26, Z 377.102, A -75.058, B 83.904, C 170.36, E1 0, E2 0, E3 0, E4 0}
LIN {X 524.985, Y 313.107, Z 376.476, A -75.058, B 83.904, C 170.36, E1 0, E2 0, E3 0, E4 0}
LIN {X 525.22, Y 308.113, Z 376.998, A -75.058, B 83.904, C 170.36, E1 0, E2 0, E3 0, E4 0}
LIN {X 552.492, Y 311.07, Z 377.443, A -75.058, B 83.904, C 170.36, E1 0, E2 0, E3 0, E4 0}
LIN {X 529.62, Y 303.569, Z 377.588, A -75.058, B 83.904, C 170.36, E1 0, E2 0, E3 0, E4 0}
LIN {X 525.302, Y 303.101, Z 377.517, A -75.058, B 83.904, C 170.36, E1 0, E2 0, E3 0, E4 0}
LIN {X 525.241, Y 365.335, Z 371.094, A -75.058, B 83.904, C 170.36, E1 0, E2 0, E3 0, E4 0}
LIN {X 525.645, Y 359.357, Z 371.722, A -75.058, B 83.904, C 170.36, E1 0, E2 0, E3 0, E4 0}
LIN {X 525.989, Y 345.052, Z 373.207, A -75.058, B 83.904, C 170.36, E1 0, E2 0, E3 0, E4 0}
LIN {X 525.628, Y 340.179, Z 373.7, A -75.058, B 83.904, C 170.36, E1 0, E2 0, E3 0, E4 0}
LIN {X 526.024, Y 338.585, Z 373.876, A -75.058, B 83.904, C 170.36, E1 0, E2 0, E3 0, E4 0}
LIN {X 525.94, Y 337.558, Z 373.979, A -75.058, B 83.904, C 170.36, E1 0, E2 0, E3 0, E4 0}
LIN {X 525.906, Y 337.49, Z 373.985, A -75.058, B 83.904, C 170.36, E1 0, E2 0, E3 0, E4 0}
LIN {X 526.257, Y 324.07, Z 375.38, A -75.058, B 83.904, C 170.36, E1 0, E2 0, E3 0, E4 0}
LIN {X 526.18, Y 323.91, Z 375.394, A -75.058, B 83.904, C 170.36, E1 0, E2 0, E3 0, E4 0}
LIN {X 525.227, Y 318.616, Z 375.914, A -75.058, B 83.904, C 170.36, E1 0, E2 0, E3 0, E4 0}
LIN {X 525.383, Y 306.532, Z 377.165, A -75.058, B 83.904, C 170.36, E1 0, E2 0, E3 0, E4 0}
LIN {X 525.31, Y 306.275, Z 377.19, A -75.058, B 83.904, C 170.36, E1 0, E2 0, E3 0, E4 0}
LIN {X 525.348, Y 301.595, Z 377.674, A -75.058, B 83.904, C 170.36, E1 0, E2 0, E3 0, E4 0}
LIN {X 564.523, Y 314.506, Z 377.42, A -75.058, B 83.904, C 170.36, E1 0, E2 0, E3 0, E4 0}
LIN {X 530.936, Y 392.041, Z 368.495, A -75.058, B 83.904, C 170.36, E1 0, E2 0, E3 0, E4 0}
LIN {X 528.78, Y 391.459, Z 368.496, A -75.058, B 83.904, C 170.36, E1 0, E2 0, E3 0, E4 0}
LIN {X 528.743, Y 391.392, Z 368.501, A -75.058, B 83.904, C 170.36, E1 0, E2 0, E3 0, E4 0}
LIN {X 527.951, Y 391.24, Z 368.495, A -75.058, B 83.904, C 170.36, E1 0, E2 0, E3 0, E4 0}
LIN {X 527.502, Y 391.304, Z 368.477, A -75.058, B 83.904, C 170.36, E1 0, E2 0, E3 0, E4 0}
LIN {X 527.469, Y 391.416, Z 368.464, A -75.058, B 83.904, C 170.36, E1 0, E2 0, E3 0, E4 0}
LIN {X 526.066, Y 391.712, Z 368.395, A -75.058, B 83.904, C 170.36, E1 0, E2 0, E3 0, E4 0}
LIN {X 523.623, Y 390.957, Z 368.405, A -75.058, B 83.904, C 170.36, E1 0, E2 0, E3 0, E4 0}
LIN {X 523.002, Y 390.946, Z 368.389, A -75.058, B 83.904, C 170.36, E1 0, E2 0, E3 0, E4 0}
LIN {X 522.565, Y 390.444, Z 368.429, A -75.058, B 83.904, C 170.36, E1 0, E2 0, E3 0, E4 0}
LIN {X 522.273, Y 389.211, Z 368.548, A -75.058, B 83.904, C 170.36, E1 0, E2 0, E3 0, E4 0}
LIN {X 524.167, Y 385.569, Z 368.976, A -75.058, B 83.904, C 170.36, E1 0, E2 0, E3 0, E4 0}
LIN {X 524.109, Y 381.847, Z 369.359, A -75.058, B 83.904, C 170.36, E1 0, E2 0, E3 0, E4 0}
LIN {X 524.395, Y 377.83, Z 369.781, A -75.058, B 83.904, C 170.36, E1 0, E2 0, E3 0, E4 0}
LIN {X 525.241, Y 365.335, Z 371.094, A -75.058, B 83.904, C 170.36, E1 0, E2 0, E3 0, E4 0}
PTP {X 532.274, Y 389.769, Z 429.374, A -75.058, B 83.904, C 170.36, E1 0, E2 0, E3 0, E4 0, S 'B010'}
PTP {A1 5, A2 -90, A3 100, A4 5, A5 -10, A6 -5, E1 0, E2 0, E3 0, E4 0} C_PTP

END
